LIN {X 0,Y 256.268,Z 255.065,A -85,B 0,C 180,E1 -18646.324,E2 -18646.324} C_VEL
LIN {X 0,Y 256.169,Z 255.063,A -85,B 0,C 180,E1 -18651.153,E2 -18651.153} C_VEL
LIN {X 0,Y 256.159,Z 255.045,A -85,B 0,C 180,E1 -18655.146,E2 -18655.146} C_VEL
LIN {X 0,Y 256.122,Z 255.064,A -85,B 0,C 180,E1 -18659.598,E2 -18659.598} C_VEL
LIN {X 0,Y 256.095,Z 255.082,A -85,B 0,C 180,E1 -18663.288,E2 -18663.288} C_VEL
LIN {X 0,Y 256.131,Z 255.076,A -85,B 0,C 180,E1 -18667.291,E2 -18667.291} C_VEL
LIN {X 0,Y 256.137,Z 255.062,A -85,B 0,C 180,E1 -18671.186,E2 -18671.186} C_VEL
LIN {X 0,Y 256.089,Z 255.082,A -85,B 0,C 180,E1 -18675.522,E2 -18675.522} C_VEL
LIN {X 0,Y 256.106,Z 255.073,A -85,B 0,C 180,E1 -18678.818,E2 -18678.818} C_VEL
LIN {X 0,Y 256.13,Z 255.056,A -85,B 0,C 180,E1 -18682.878,E2 -18682.878} C_VEL
LIN {X 0,Y 256.062,Z 255.088,A -85,B 0,C 180,E1 -18686.717,E2 -18686.717} C_VEL
LIN {X 0,Y 256.118,Z 255.044,A -85,B 0,C 180,E1 -18691.412,E2 -18691.412} C_VEL
LIN {X 0,Y 256.151,Z 255.067,A -85,B 0,C 180,E1 -18695.706,E2 -18695.706} C_VEL
LIN {X 0,Y 256.218,Z 255.067,A -85,B 0,C 180,E1 -18699.118,E2 -18699.118} C_VEL
LIN {X 0,Y 256.282,Z 255.016,A -85,B 0,C 180,E1 -18704.092,E2 -18704.092} C_VEL
LIN {X 0,Y 256.301,Z 255.048,A -85,B 0,C 180,E1 -18708.941,E2 -18708.941} C_VEL
LIN {X 0,Y 256.533,Z 255.027,A -85,B 0,C 180,E1 -18712.134,E2 -18712.134} C_VEL
LIN {X 0,Y 256.71,Z 254.962,A -85,B 0,C 180,E1 -18718.438,E2 -18718.438} C_VEL
LIN {X 0,Y 256.736,Z 254.971,A -85,B 0,C 180,E1 -18719.772,E2 -18719.772} C_VEL
LIN {X 0,Y 256.465,Z 255.019,A -85,B 0,C 180,E1 -18720.645,E2 -18720.645} C_VEL
LIN {X 0,Y 255.123,Z 255.201,A -85,B 0,C 180,E1 -18721.933,E2 -18721.933} C_VEL
LIN {X 0,Y 250.65,Z 255.767,A -85,B 0,C 180,E1 -18724.929,E2 -18724.929} C_VEL
LIN {X 0,Y 249.524,Z 255.896,A -85,B 0,C 180,E1 -18726.273,E2 -18726.273} C_VEL
LIN {X 0,Y 249.417,Z 255.903,A -85,B 0,C 180,E1 -18726.73,E2 -18726.73} C_VEL
LIN {X 0,Y 249.345,Z 255.885,A -85,B 0,C 180,E1 -18729.743,E2 -18729.743} C_VEL
LIN {X 0,Y 249.21,Z 255.942,A -85,B 0,C 180,E1 -18734.71,E2 -18734.71} C_VEL
LIN {X 0,Y 249.144,Z 255.941,A -85,B 0,C 180,E1 -18738.084,E2 -18738.084} C_VEL
LIN {X 0,Y 249.091,Z 255.926,A -85,B 0,C 180,E1 -18741.524,E2 -18741.524} C_VEL
LIN {X 0,Y 249.125,Z 255.954,A -85,B 0,C 180,E1 -18745.481,E2 -18745.481} C_VEL
LIN {X 0,Y 249.065,Z 255.939,A -85,B 0,C 180,E1 -18748.987,E2 -18748.987} C_VEL
LIN {X 0,Y 249.038,Z 255.962,A -85,B 0,C 180,E1 -18752.432,E2 -18752.432} C_VEL
LIN {X 0,Y 249.038,Z 255.952,A -85,B 0,C 180,E1 -18756.351,E2 -18756.351} C_VEL
LIN {X 0,Y 249.019,Z 255.966,A -85,B 0,C 180,E1 -18760.483,E2 -18760.483} C_VEL
LIN {X 0,Y 249.014,Z 255.942,A -85,B 0,C 180,E1 -18762.795,E2 -18762.795} C_VEL
LIN {X 0,Y 248.992,Z 255.944,A -85,B 0,C 180,E1 -18767.359,E2 -18767.359} C_VEL
LIN {X 0,Y 249.017,Z 255.952,A -85,B 0,C 180,E1 -18771.619,E2 -18771.619} C_VEL
LIN {X 0,Y 249.109,Z 256,A -85,B 0,C 180,E1 -18776.504,E2 -18776.504} C_VEL
LIN {X 0,Y 251.031,Z 265.205,A -85,B 0,C 180,E1 -18780.224,E2 -18780.224} C_VEL
LIN {X 0,Y 251.514,Z 267.303,A -85,B 0,C 180,E1 -18780.91,E2 -18780.91} C_VEL
LIN {X 0,Y 257.248,Z 283.893,A -85,B 0,C 180,E1 -18782.001,E2 -18782.001} C_VEL
LIN {X 0,Y 261.027,Z 311.595,A -85,B 0,C 180,E1 -18783.167,E2 -18783.167} C_VEL
LIN {X 0,Y 259.211,Z 375.113,A -85,B 0,C 180,E1 -18784.936,E2 -18784.936} C_VEL
LIN {X 0,Y 258.333,Z 387.52,A -85,B 0,C 180,E1 -18785.543,E2 -18785.543} C_VEL
LIN {X 0,Y 257.11,Z 401.037,A -85,B 0,C 180,E1 -18786.544,E2 -18786.544} C_VEL
LIN {X 0,Y 255.546,Z 413.128,A -85,B 0,C 180,E1 -18787.781,E2 -18787.781} C_VEL
LIN {X 0,Y 253.899,Z 424.693,A -85,B 0,C 180,E1 -18789.334,E2 -18789.334} C_VEL
LIN {X 0,Y 252.383,Z 435.261,A -85,B 0,C 180,E1 -18791.141,E2 -18791.141} C_VEL
LIN {X 0,Y 250.81,Z 445.277,A -85,B 0,C 180,E1 -18793.309,E2 -18793.309} C_VEL
LIN {X 0,Y 249.345,Z 454.181,A -85,B 0,C 180,E1 -18795.723,E2 -18795.723} C_VEL
LIN {X 0,Y 248.261,Z 461.278,A -85,B 0,C 180,E1 -18798.157,E2 -18798.157} C_VEL
LIN {X 0,Y 247.426,Z 467.749,A -85,B 0,C 180,E1 -18801.013,E2 -18801.013} C_VEL
LIN {X 0,Y 247.028,Z 471.99,A -85,B 0,C 180,E1 -18803.466,E2 -18803.466} C_VEL
LIN {X 0,Y 246.86,Z 474.371,A -85,B 0,C 180,E1 -18805.217,E2 -18805.217} C_VEL
LIN {X 0,Y 246.839,Z 475.983,A -85,B 0,C 180,E1 -18806.736,E2 -18806.736} C_VEL
LIN {X 0,Y 246.87,Z 477.31,A -85,B 0,C 180,E1 -18808.369,E2 -18808.369} C_VEL
LIN {X 0,Y 246.903,Z 478.239,A -85,B 0,C 180,E1 -18810.001,E2 -18810.001} C_VEL
LIN {X 0,Y 246.87,Z 478.771,A -85,B 0,C 180,E1 -18811.632,E2 -18811.632} C_VEL
LIN {X 0,Y 246.942,Z 478.586,A -85,B 0,C 180,E1 -18814.898,E2 -18814.898} C_VEL
LIN {X 0,Y 247.422,Z 476.873,A -85,B 0,C 180,E1 -18818.166,E2 -18818.166} C_VEL
LIN {X 0,Y 247.888,Z 475.394,A -85,B 0,C 180,E1 -18819.795,E2 -18819.795} C_VEL
LIN {X 0,Y 248.918,Z 472.402,A -85,B 0,C 180,E1 -18822.226,E2 -18822.226} C_VEL
LIN {X 0,Y 250.251,Z 468.389,A -85,B 0,C 180,E1 -18824.641,E2 -18824.641} C_VEL
LIN {X 0,Y 252.491,Z 462.242,A -85,B 0,C 180,E1 -18827.411,E2 -18827.411} C_VEL
LIN {X 0,Y 254.814,Z 455.623,A -85,B 0,C 180,E1 -18829.73,E2 -18829.73} C_VEL
LIN {X 0,Y 257.32,Z 447.491,A -85,B 0,C 180,E1 -18832.016,E2 -18832.016} C_VEL
LIN {X 0,Y 259.942,Z 438.896,A -85,B 0,C 180,E1 -18833.926,E2 -18833.926} C_VEL
LIN {X 0,Y 262.902,Z 428.491,A -85,B 0,C 180,E1 -18835.748,E2 -18835.748} C_VEL
LIN {X 0,Y 265.736,Z 416.819,A -85,B 0,C 180,E1 -18837.357,E2 -18837.357} C_VEL
LIN {X 0,Y 268.156,Z 405.109,A -85,B 0,C 180,E1 -18838.575,E2 -18838.575} C_VEL
LIN {X 0,Y 270.132,Z 393.004,A -85,B 0,C 180,E1 -18839.518,E2 -18839.518} C_VEL
LIN {X 0,Y 271.689,Z 379.85,A -85,B 0,C 180,E1 -18840.239,E2 -18840.239} C_VEL
LIN {X 0,Y 272.619,Z 364.907,A -85,B 0,C 180,E1 -18840.726,E2 -18840.726} C_VEL
LIN {X 0,Y 274.682,Z 317.162,A -85,B 0,C 180,E1 -18841.977,E2 -18841.977} C_VEL
LIN {X 0,Y 272.652,Z 306.034,A -85,B 0,C 180,E1 -18842.686,E2 -18842.686} C_VEL
LIN {X 0,Y 266.598,Z 292.603,A -85,B 0,C 180,E1 -18844.214,E2 -18844.214} C_VEL
LIN {X 0,Y 257.687,Z 275.866,A -85,B 0,C 180,E1 -18846.542,E2 -18846.542} C_VEL
LIN {X 0,Y 254.296,Z 270.358,A -85,B 0,C 180,E1 -18847.462,E2 -18847.462} C_VEL
LIN {X 0,Y 251.99,Z 266.272,A -85,B 0,C 180,E1 -18848.205,E2 -18848.205} C_VEL
LIN {X 0,Y 249.946,Z 259.327,A -85,B 0,C 180,E1 -18851.822,E2 -18851.822} C_VEL
LIN {X 0,Y 249.003,Z 255.983,A -85,B 0,C 180,E1 -18853.876,E2 -18853.876} C_VEL
LIN {X 0,Y 249.022,Z 255.94,A -85,B 0,C 180,E1 -18857.357,E2 -18857.357} C_VEL
LIN {X 0,Y 249.056,Z 255.957,A -85,B 0,C 180,E1 -18862.197,E2 -18862.197} C_VEL
LIN {X 0,Y 249.058,Z 255.959,A -85,B 0,C 180,E1 -18865.635,E2 -18865.635} C_VEL
LIN {X 0,Y 249.015,Z 255.966,A -85,B 0,C 180,E1 -18869.461,E2 -18869.461} C_VEL
LIN {X 0,Y 249.028,Z 255.962,A -85,B 0,C 180,E1 -18873.15,E2 -18873.15} C_VEL
LIN {X 0,Y 249.017,Z 255.959,A -85,B 0,C 180,E1 -18876.72,E2 -18876.72} C_VEL
LIN {X 0,Y 249.068,Z 255.947,A -85,B 0,C 180,E1 -18880.201,E2 -18880.201} C_VEL
LIN {X 0,Y 249.186,Z 255.935,A -85,B 0,C 180,E1 -18883.611,E2 -18883.611} C_VEL
LIN {X 0,Y 249.245,Z 255.926,A -85,B 0,C 180,E1 -18888.609,E2 -18888.609} C_VEL
LIN {X 0,Y 249.445,Z 255.913,A -85,B 0,C 180,E1 -18891.895,E2 -18891.895} C_VEL
LIN {X 0,Y 249.277,Z 255.928,A -85,B 0,C 180,E1 -18895.141,E2 -18895.141} C_VEL
LIN {X 0,Y 249.666,Z 255.872,A -85,B 0,C 180,E1 -18898.38,E2 -18898.38} C_VEL
LIN {X 0,Y 249.671,Z 255.881,A -85,B 0,C 180,E1 -18901.606,E2 -18901.606} C_VEL
LIN {X 0,Y 249.425,Z 255.906,A -85,B 0,C 180,E1 -18906.532,E2 -18906.532} C_VEL
LIN {X 0,Y 249.34,Z 255.927,A -85,B 0,C 180,E1 -18909.729,E2 -18909.729} C_VEL
LIN {X 0,Y 249.176,Z 255.939,A -85,B 0,C 180,E1 -18914.697,E2 -18914.697} C_VEL
LIN {X 0,Y 249.111,Z 255.949,A -85,B 0,C 180,E1 -18918.071,E2 -18918.071} C_VEL
LIN {X 0,Y 249.076,Z 255.953,A -85,B 0,C 180,E1 -18921.51,E2 -18921.51} C_VEL
LIN {X 0,Y 249.116,Z 255.93,A -85,B 0,C 180,E1 -18925.474,E2 -18925.474} C_VEL
LIN {X 0,Y 249.033,Z 255.949,A -85,B 0,C 180,E1 -18930.095,E2 -18930.095} C_VEL
LIN {X 0,Y 249.056,Z 256.275,A -85,B 0,C 180,E1 -18930.751,E2 -18930.751} C_VEL
LIN {X 0,Y 250.702,Z 261.422,A -85,B 0,C 180,E1 -18933.56,E2 -18933.56} C_VEL
LIN {X 0,Y 253.421,Z 265.892,A -85,B 0,C 180,E1 -18934.408,E2 -18934.408} C_VEL
LIN {X 0,Y 259.859,Z 276.539,A -85,B 0,C 180,E1 -18936.154,E2 -18936.154} C_VEL
LIN {X 0,Y 266.04,Z 287.62,A -85,B 0,C 180,E1 -18937.741,E2 -18937.741} C_VEL
LIN {X 0,Y 273.058,Z 302.502,A -85,B 0,C 180,E1 -18939.498,E2 -18939.498} C_VEL
LIN {X 0,Y 275.043,Z 307.322,A -85,B 0,C 180,E1 -18939.99,E2 -18939.99} C_VEL
LIN {X 0,Y 272.309,Z 368.99,A -85,B 0,C 180,E1 -18941.647,E2 -18941.647} C_VEL
LIN {X 0,Y 271.045,Z 381.678,A -85,B 0,C 180,E1 -18942.233,E2 -18942.233} C_VEL
LIN {X 0,Y 269.395,Z 393.837,A -85,B 0,C 180,E1 -18943.074,E2 -18943.074} C_VEL
LIN {X 0,Y 267.158,Z 405.932,A -85,B 0,C 180,E1 -18944.204,E2 -18944.204} C_VEL
LIN {X 0,Y 264.797,Z 416.671,A -85,B 0,C 180,E1 -18945.531,E2 -18945.531} C_VEL
LIN {X 0,Y 261.869,Z 428.103,A -85,B 0,C 180,E1 -18947.339,E2 -18947.339} C_VEL
LIN {X 0,Y 258.942,Z 438.019,A -85,B 0,C 180,E1 -18949.353,E2 -18949.353} C_VEL
LIN {X 0,Y 256.367,Z 446.072,A -85,B 0,C 180,E1 -18951.415,E2 -18951.415} C_VEL
LIN {X 0,Y 253.816,Z 453.448,A -85,B 0,C 180,E1 -18953.782,E2 -18953.782} C_VEL
LIN {X 0,Y 251.804,Z 459.061,A -85,B 0,C 180,E1 -18956.067,E2 -18956.067} C_VEL
LIN {X 0,Y 249.967,Z 464.011,A -85,B 0,C 180,E1 -18958.658,E2 -18958.658} C_VEL
LIN {X 0,Y 248.598,Z 467.684,A -85,B 0,C 180,E1 -18961.275,E2 -18961.275} C_VEL
LIN {X 0,Y 247.898,Z 469.469,A -85,B 0,C 180,E1 -18963.024,E2 -18963.024} C_VEL
LIN {X 0,Y 247.242,Z 471.174,A -85,B 0,C 180,E1 -18965.429,E2 -18965.429} C_VEL
LIN {X 0,Y 246.716,Z 472.063,A -85,B 0,C 180,E1 -18968.264,E2 -18968.264} C_VEL
LIN {X 0,Y 246.593,Z 472.02,A -85,B 0,C 180,E1 -18970.109,E2 -18970.109} C_VEL
LIN {X 0,Y 246.5,Z 471.576,A -85,B 0,C 180,E1 -18971.722,E2 -18971.722} C_VEL
LIN {X 0,Y 246.481,Z 470.644,A -85,B 0,C 180,E1 -18973.433,E2 -18973.433} C_VEL
LIN {X 0,Y 246.665,Z 468.876,A -85,B 0,C 180,E1 -18975.594,E2 -18975.594} C_VEL
LIN {X 0,Y 247.089,Z 465.228,A -85,B 0,C 180,E1 -18978.515,E2 -18978.515} C_VEL
LIN {X 0,Y 247.589,Z 460.912,A -85,B 0,C 180,E1 -18981.018,E2 -18981.018} C_VEL
LIN {X 0,Y 248.411,Z 455.369,A -85,B 0,C 180,E1 -18983.502,E2 -18983.502} C_VEL
LIN {X 0,Y 249.424,Z 448.448,A -85,B 0,C 180,E1 -18985.96,E2 -18985.96} C_VEL
LIN {X 0,Y 250.55,Z 441.374,A -85,B 0,C 180,E1 -18987.99,E2 -18987.99} C_VEL
LIN {X 0,Y 251.912,Z 432.846,A -85,B 0,C 180,E1 -18989.999,E2 -18989.999} C_VEL
LIN {X 0,Y 253.636,Z 422.254,A -85,B 0,C 180,E1 -18991.984,E2 -18991.984} C_VEL
LIN {X 0,Y 255.344,Z 410.323,A -85,B 0,C 180,E1 -18993.747,E2 -18993.747} C_VEL
LIN {X 0,Y 256.801,Z 398.302,A -85,B 0,C 180,E1 -18995.102,E2 -18995.102} C_VEL
LIN {X 0,Y 257.943,Z 385.834,A -85,B 0,C 180,E1 -18996.158,E2 -18996.158} C_VEL
LIN {X 0,Y 258.952,Z 372.79,A -85,B 0,C 180,E1 -18996.917,E2 -18996.917} C_VEL
LIN {X 0,Y 259.526,Z 357.393,A -85,B 0,C 180,E1 -18997.439,E2 -18997.439} C_VEL
LIN {X 0,Y 261.24,Z 299.46,A -85,B 0,C 180,E1 -18999.006,E2 -18999.006} C_VEL
LIN {X 0,Y 259.014,Z 285.584,A -85,B 0,C 180,E1 -18999.617,E2 -18999.617} C_VEL
LIN {X 0,Y 253.614,Z 269.571,A -85,B 0,C 180,E1 -19000.609,E2 -19000.609} C_VEL
LIN {X 0,Y 250.347,Z 261.084,A -85,B 0,C 180,E1 -19001.239,E2 -19001.239} C_VEL
LIN {X 0,Y 249.257,Z 256.073,A -85,B 0,C 180,E1 -19003.191,E2 -19003.191} C_VEL
LIN {X 0,Y 249.21,Z 255.943,A -85,B 0,C 180,E1 -19006.531,E2 -19006.531} C_VEL
LIN {X 0,Y 249.103,Z 255.948,A -85,B 0,C 180,E1 -19011.516,E2 -19011.516} C_VEL
LIN {X 0,Y 249.1,Z 255.918,A -85,B 0,C 180,E1 -19015.489,E2 -19015.489} C_VEL
LIN {X 0,Y 249.099,Z 255.929,A -85,B 0,C 180,E1 -19019.019,E2 -19019.019} C_VEL
LIN {X 0,Y 249.039,Z 255.966,A -85,B 0,C 180,E1 -19022.424,E2 -19022.424} C_VEL
LIN {X 0,Y 249.061,Z 255.95,A -85,B 0,C 180,E1 -19026.339,E2 -19026.339} C_VEL
LIN {X 0,Y 249.104,Z 255.947,A -85,B 0,C 180,E1 -19030.458,E2 -19030.458} C_VEL
LIN {X 0,Y 249.035,Z 255.959,A -85,B 0,C 180,E1 -19034.871,E2 -19034.871} C_VEL
LIN {X 0,Y 249.071,Z 255.959,A -85,B 0,C 180,E1 -19037.387,E2 -19037.387} C_VEL
LIN {X 0,Y 249.027,Z 255.931,A -85,B 0,C 180,E1 -19041.631,E2 -19041.631} C_VEL
LIN {X 0,Y 249.038,Z 255.961,A -85,B 0,C 180,E1 -19045.649,E2 -19045.649} C_VEL
LIN {X 0,Y 249.031,Z 255.95,A -85,B 0,C 180,E1 -19049.48,E2 -19049.48} C_VEL
LIN {X 0,Y 249.055,Z 255.922,A -85,B 0,C 180,E1 -19053.17,E2 -19053.17} C_VEL
LIN {X 0,Y 249.071,Z 255.954,A -85,B 0,C 180,E1 -19056.741,E2 -19056.741} C_VEL
LIN {X 0,Y 249.132,Z 255.948,A -85,B 0,C 180,E1 -19060.222,E2 -19060.222} C_VEL
LIN {X 0,Y 249.23,Z 255.897,A -85,B 0,C 180,E1 -19063.629,E2 -19063.629} C_VEL
LIN {X 0,Y 249.244,Z 255.925,A -85,B 0,C 180,E1 -19068.624,E2 -19068.624} C_VEL
LIN {X 0,Y 249.477,Z 255.906,A -85,B 0,C 180,E1 -19071.91,E2 -19071.91} C_VEL
LIN {X 0,Y 249.43,Z 255.871,A -85,B 0,C 180,E1 -19076.777,E2 -19076.777} C_VEL
LIN {X 0,Y 249.718,Z 255.848,A -85,B 0,C 180,E1 -19080.007,E2 -19080.007} C_VEL
LIN {X 0,Y 249.43,Z 255.912,A -85,B 0,C 180,E1 -19083.238,E2 -19083.238} C_VEL
LIN {X 0,Y 249.417,Z 255.903,A -85,B 0,C 180,E1 -19086.73,E2 -19086.73} C_VEL
LIN {X 0,Y 248.696,Z 255.981,A -85,B 0,C 180,E1 -19088.076,E2 -19088.076} C_VEL
LIN {X 0,Y 245.771,Z 256.344,A -85,B 0,C 180,E1 -19090.268,E2 -19090.268} C_VEL
LIN {X 0,Y 243.304,Z 256.66,A -85,B 0,C 180,E1 -19092.054,E2 -19092.054} C_VEL
LIN {X 0,Y 242.237,Z 256.8,A -85,B 0,C 180,E1 -19093.441,E2 -19093.441} C_VEL
LIN {X 0,Y 242.145,Z 256.811,A -85,B 0,C 180,E1 -19093.911,E2 -19093.911} C_VEL
LIN {X 0,Y 242.156,Z 256.818,A -85,B 0,C 180,E1 -19096.878,E2 -19096.878} C_VEL
LIN {X 0,Y 242.033,Z 256.806,A -85,B 0,C 180,E1 -19101.693,E2 -19101.693} C_VEL
LIN {X 0,Y 242.076,Z 256.832,A -85,B 0,C 180,E1 -19105.844,E2 -19105.844} C_VEL
LIN {X 0,Y 241.986,Z 256.818,A -85,B 0,C 180,E1 -19109.593,E2 -19109.593} C_VEL
LIN {X 0,Y 241.99,Z 256.846,A -85,B 0,C 180,E1 -19113.498,E2 -19113.498} C_VEL
LIN {X 0,Y 241.995,Z 256.826,A -85,B 0,C 180,E1 -19117.588,E2 -19117.588} C_VEL
LIN {X 0,Y 241.947,Z 256.838,A -85,B 0,C 180,E1 -19121.928,E2 -19121.928} C_VEL
LIN {X 0,Y 241.916,Z 256.811,A -85,B 0,C 180,E1 -19126.584,E2 -19126.584} C_VEL
LIN {X 0,Y 241.944,Z 256.844,A -85,B 0,C 180,E1 -19130.28,E2 -19130.28} C_VEL
LIN {X 0,Y 241.989,Z 256.841,A -85,B 0,C 180,E1 -19134.49,E2 -19134.49} C_VEL
LIN {X 0,Y 242.088,Z 257.038,A -85,B 0,C 180,E1 -19136.15,E2 -19136.15} C_VEL
LIN {X 0,Y 244.179,Z 266.965,A -85,B 0,C 180,E1 -19140.133,E2 -19140.133} C_VEL
LIN {X 0,Y 246.952,Z 274.593,A -85,B 0,C 180,E1 -19140.729,E2 -19140.729} C_VEL
LIN {X 0,Y 250.974,Z 286.669,A -85,B 0,C 180,E1 -19141.497,E2 -19141.497} C_VEL
LIN {X 0,Y 254.446,Z 312.616,A -85,B 0,C 180,E1 -19142.618,E2 -19142.618} C_VEL
LIN {X 0,Y 252.549,Z 374.939,A -85,B 0,C 180,E1 -19144.393,E2 -19144.393} C_VEL
LIN {X 0,Y 251.653,Z 387.375,A -85,B 0,C 180,E1 -19145.014,E2 -19145.014} C_VEL
LIN {X 0,Y 250.447,Z 400.339,A -85,B 0,C 180,E1 -19145.991,E2 -19145.991} C_VEL
LIN {X 0,Y 248.968,Z 411.809,A -85,B 0,C 180,E1 -19147.162,E2 -19147.162} C_VEL
LIN {X 0,Y 247.192,Z 423.597,A -85,B 0,C 180,E1 -19148.747,E2 -19148.747} C_VEL
LIN {X 0,Y 245.658,Z 434.253,A -85,B 0,C 180,E1 -19150.584,E2 -19150.584} C_VEL
LIN {X 0,Y 244.328,Z 442.864,A -85,B 0,C 180,E1 -19152.421,E2 -19152.421} C_VEL
LIN {X 0,Y 242.933,Z 450.808,A -85,B 0,C 180,E1 -19154.479,E2 -19154.479} C_VEL
LIN {X 0,Y 241.563,Z 458.535,A -85,B 0,C 180,E1 -19156.97,E2 -19156.97} C_VEL
LIN {X 0,Y 240.842,Z 463.824,A -85,B 0,C 180,E1 -19159.067,E2 -19159.067} C_VEL
LIN {X 0,Y 240.224,Z 468.923,A -85,B 0,C 180,E1 -19161.589,E2 -19161.589} C_VEL
LIN {X 0,Y 239.847,Z 472.858,A -85,B 0,C 180,E1 -19164.114,E2 -19164.114} C_VEL
LIN {X 0,Y 239.746,Z 475.746,A -85,B 0,C 180,E1 -19166.639,E2 -19166.639} C_VEL
LIN {X 0,Y 239.784,Z 477.105,A -85,B 0,C 180,E1 -19168.321,E2 -19168.321} C_VEL
LIN {X 0,Y 239.816,Z 478.064,A -85,B 0,C 180,E1 -19170.001,E2 -19170.001} C_VEL
LIN {X 0,Y 239.784,Z 478.631,A -85,B 0,C 180,E1 -19171.68,E2 -19171.68} C_VEL
LIN {X 0,Y 239.855,Z 478.57,A -85,B 0,C 180,E1 -19174.916,E2 -19174.916} C_VEL
LIN {X 0,Y 240.055,Z 477.898,A -85,B 0,C 180,E1 -19176.726,E2 -19176.726} C_VEL
LIN {X 0,Y 240.894,Z 475.469,A -85,B 0,C 180,E1 -19180.082,E2 -19180.082} C_VEL
LIN {X 0,Y 241.975,Z 472.536,A -85,B 0,C 180,E1 -19182.582,E2 -19182.582} C_VEL
LIN {X 0,Y 243.372,Z 468.589,A -85,B 0,C 180,E1 -19185.065,E2 -19185.065} C_VEL
LIN {X 0,Y 245.398,Z 463.528,A -85,B 0,C 180,E1 -19187.501,E2 -19187.501} C_VEL
LIN {X 0,Y 247.768,Z 457.187,A -85,B 0,C 180,E1 -19189.901,E2 -19189.901} C_VEL
LIN {X 0,Y 250.209,Z 449.606,A -85,B 0,C 180,E1 -19192.197,E2 -19192.197} C_VEL
LIN {X 0,Y 252.952,Z 441.298,A -85,B 0,C 180,E1 -19194.193,E2 -19194.193} C_VEL
LIN {X 0,Y 255.966,Z 431.541,A -85,B 0,C 180,E1 -19196.06,E2 -19196.06} C_VEL
LIN {X 0,Y 258.874,Z 420.66,A -85,B 0,C 180,E1 -19197.705,E2 -19197.705} C_VEL
LIN {X 0,Y 261.315,Z 410.047,A -85,B 0,C 180,E1 -19198.954,E2 -19198.954} C_VEL
LIN {X 0,Y 263.489,Z 398.442,A -85,B 0,C 180,E1 -19200.008,E2 -19200.008} C_VEL
LIN {X 0,Y 265.39,Z 385.352,A -85,B 0,C 180,E1 -19200.867,E2 -19200.867} C_VEL
LIN {X 0,Y 266.579,Z 372.119,A -85,B 0,C 180,E1 -19201.427,E2 -19201.427} C_VEL
LIN {X 0,Y 269.08,Z 318.313,A -85,B 0,C 180,E1 -19202.874,E2 -19202.874} C_VEL
LIN {X 0,Y 267.46,Z 309.167,A -85,B 0,C 180,E1 -19203.475,E2 -19203.475} C_VEL
LIN {X 0,Y 261.518,Z 296.019,A -85,B 0,C 180,E1 -19205.04,E2 -19205.04} C_VEL
LIN {X 0,Y 253.419,Z 280.618,A -85,B 0,C 180,E1 -19207.254,E2 -19207.254} C_VEL
LIN {X 0,Y 249.605,Z 274.39,A -85,B 0,C 180,E1 -19208.34,E2 -19208.34} C_VEL
LIN {X 0,Y 247.069,Z 270.251,A -85,B 0,C 180,E1 -19209.102,E2 -19209.102} C_VEL
LIN {X 0,Y 244.678,Z 266.104,A -85,B 0,C 180,E1 -19209.931,E2 -19209.931} C_VEL
LIN {X 0,Y 242.716,Z 259.494,A -85,B 0,C 180,E1 -19213.615,E2 -19213.615} C_VEL
LIN {X 0,Y 241.944,Z 256.873,A -85,B 0,C 180,E1 -19215.396,E2 -19215.396} C_VEL
LIN {X 0,Y 241.935,Z 256.835,A -85,B 0,C 180,E1 -19219.05,E2 -19219.05} C_VEL
LIN {X 0,Y 241.999,Z 256.838,A -85,B 0,C 180,E1 -19222.413,E2 -19222.413} C_VEL
LIN {X 0,Y 241.994,Z 256.843,A -85,B 0,C 180,E1 -19226.502,E2 -19226.502} C_VEL
LIN {X 0,Y 241.989,Z 256.837,A -85,B 0,C 180,E1 -19230.608,E2 -19230.608} C_VEL
LIN {X 0,Y 242.008,Z 256.839,A -85,B 0,C 180,E1 -19234.192,E2 -19234.192} C_VEL
LIN {X 0,Y 241.997,Z 256.841,A -85,B 0,C 180,E1 -19238.332,E2 -19238.332} C_VEL
LIN {X 0,Y 242.125,Z 256.817,A -85,B 0,C 180,E1 -19243.31,E2 -19243.31} C_VEL
LIN {X 0,Y 242.18,Z 256.808,A -85,B 0,C 180,E1 -19248.272,E2 -19248.272} C_VEL
LIN {X 0,Y 242.394,Z 256.793,A -85,B 0,C 180,E1 -19251.657,E2 -19251.657} C_VEL
LIN {X 0,Y 242.238,Z 256.803,A -85,B 0,C 180,E1 -19254.999,E2 -19254.999} C_VEL
LIN {X 0,Y 242.625,Z 256.749,A -85,B 0,C 180,E1 -19258.333,E2 -19258.333} C_VEL
LIN {X 0,Y 242.632,Z 256.757,A -85,B 0,C 180,E1 -19261.652,E2 -19261.652} C_VEL
LIN {X 0,Y 242.399,Z 256.78,A -85,B 0,C 180,E1 -19266.652,E2 -19266.652} C_VEL
LIN {X 0,Y 242.264,Z 256.805,A -85,B 0,C 180,E1 -19270.016,E2 -19270.016} C_VEL
LIN {X 0,Y 242.132,Z 256.814,A -85,B 0,C 180,E1 -19275.135,E2 -19275.135} C_VEL
LIN {X 0,Y 242.05,Z 256.826,A -85,B 0,C 180,E1 -19278.617,E2 -19278.617} C_VEL
LIN {X 0,Y 242.001,Z 256.833,A -85,B 0,C 180,E1 -19282.172,E2 -19282.172} C_VEL
LIN {X 0,Y 242.053,Z 256.807,A -85,B 0,C 180,E1 -19285.83,E2 -19285.83} C_VEL
LIN {X 0,Y 242.05,Z 256.877,A -85,B 0,C 180,E1 -19289.008,E2 -19289.008} C_VEL
LIN {X 0,Y 243.33,Z 261.381,A -85,B 0,C 180,E1 -19291.739,E2 -19291.739} C_VEL
LIN {X 0,Y 245.842,Z 265.498,A -85,B 0,C 180,E1 -19292.639,E2 -19292.639} C_VEL
LIN {X 0,Y 252.53,Z 275.938,A -85,B 0,C 180,E1 -19294.607,E2 -19294.607} C_VEL
LIN {X 0,Y 260.166,Z 289.495,A -85,B 0,C 180,E1 -19296.693,E2 -19296.693} C_VEL
LIN {X 0,Y 266.617,Z 302.832,A -85,B 0,C 180,E1 -19298.386,E2 -19298.386} C_VEL
LIN {X 0,Y 269.412,Z 309.425,A -85,B 0,C 180,E1 -19299.111,E2 -19299.111} C_VEL
LIN {X 0,Y 266.606,Z 369.315,A -85,B 0,C 180,E1 -19300.752,E2 -19300.752} C_VEL
LIN {X 0,Y 265.275,Z 382.204,A -85,B 0,C 180,E1 -19301.365,E2 -19301.365} C_VEL
LIN {X 0,Y 263.469,Z 394.658,A -85,B 0,C 180,E1 -19302.249,E2 -19302.249} C_VEL
LIN {X 0,Y 261.148,Z 406.518,A -85,B 0,C 180,E1 -19303.396,E2 -19303.396} C_VEL
LIN {X 0,Y 258.299,Z 418.736,A -85,B 0,C 180,E1 -19304.974,E2 -19304.974} C_VEL
LIN {X 0,Y 255.324,Z 429.583,A -85,B 0,C 180,E1 -19306.787,E2 -19306.787} C_VEL
LIN {X 0,Y 252.236,Z 439.422,A -85,B 0,C 180,E1 -19308.893,E2 -19308.893} C_VEL
LIN {X 0,Y 249.411,Z 447.817,A -85,B 0,C 180,E1 -19311.173,E2 -19311.173} C_VEL
LIN {X 0,Y 246.647,Z 455.225,A -85,B 0,C 180,E1 -19313.754,E2 -19313.754} C_VEL
LIN {X 0,Y 244.277,Z 461.337,A -85,B 0,C 180,E1 -19316.531,E2 -19316.531} C_VEL
LIN {X 0,Y 242.37,Z 466.176,A -85,B 0,C 180,E1 -19319.506,E2 -19319.506} C_VEL
LIN {X 0,Y 241.095,Z 469.234,A -85,B 0,C 180,E1 -19322.198,E2 -19322.198} C_VEL
LIN {X 0,Y 240.228,Z 471.271,A -85,B 0,C 180,E1 -19325.06,E2 -19325.06} C_VEL
LIN {X 0,Y 239.716,Z 472.129,A -85,B 0,C 180,E1 -19327.596,E2 -19327.596} C_VEL
LIN {X 0,Y 239.498,Z 472.124,A -85,B 0,C 180,E1 -19329.86,E2 -19329.86} C_VEL
LIN {X 0,Y 239.375,Z 471.003,A -85,B 0,C 180,E1 -19332.926,E2 -19332.926} C_VEL
LIN {X 0,Y 239.565,Z 469.06,A -85,B 0,C 180,E1 -19335.449,E2 -19335.449} C_VEL
LIN {X 0,Y 239.935,Z 465.888,A -85,B 0,C 180,E1 -19338.168,E2 -19338.168} C_VEL
LIN {X 0,Y 240.405,Z 461.74,A -85,B 0,C 180,E1 -19340.747,E2 -19340.747} C_VEL
LIN {X 0,Y 241.391,Z 455.34,A -85,B 0,C 180,E1 -19343.731,E2 -19343.731} C_VEL
LIN {X 0,Y 242.436,Z 448.393,A -85,B 0,C 180,E1 -19346.26,E2 -19346.26} C_VEL
LIN {X 0,Y 243.619,Z 441.287,A -85,B 0,C 180,E1 -19348.346,E2 -19348.346} C_VEL
LIN {X 0,Y 245.071,Z 432.517,A -85,B 0,C 180,E1 -19350.451,E2 -19350.451} C_VEL
LIN {X 0,Y 246.862,Z 421.841,A -85,B 0,C 180,E1 -19352.483,E2 -19352.483} C_VEL
LIN {X 0,Y 248.606,Z 410.037,A -85,B 0,C 180,E1 -19354.255,E2 -19354.255} C_VEL
LIN {X 0,Y 250.112,Z 397.885,A -85,B 0,C 180,E1 -19355.643,E2 -19355.643} C_VEL
LIN {X 0,Y 251.29,Z 385.26,A -85,B 0,C 180,E1 -19356.725,E2 -19356.725} C_VEL
LIN {X 0,Y 252.281,Z 372.846,A -85,B 0,C 180,E1 -19357.452,E2 -19357.452} C_VEL
LIN {X 0,Y 252.876,Z 357.439,A -85,B 0,C 180,E1 -19357.987,E2 -19357.987} C_VEL
LIN {X 0,Y 254.641,Z 299.96,A -85,B 0,C 180,E1 -19359.581,E2 -19359.581} C_VEL
LIN {X 0,Y 252.6,Z 287.557,A -85,B 0,C 180,E1 -19360.152,E2 -19360.152} C_VEL
LIN {X 0,Y 247.577,Z 272.582,A -85,B 0,C 180,E1 -19361.115,E2 -19361.115} C_VEL
LIN {X 0,Y 243.17,Z 261.277,A -85,B 0,C 180,E1 -19361.957,E2 -19361.957} C_VEL
LIN {X 0,Y 242.317,Z 257.497,A -85,B 0,C 180,E1 -19363.416,E2 -19363.416} C_VEL
LIN {X 0,Y 242.177,Z 256.859,A -85,B 0,C 180,E1 -19363.851,E2 -19363.851} C_VEL
LIN {X 0,Y 242.126,Z 256.821,A -85,B 0,C 180,E1 -19366.873,E2 -19366.873} C_VEL
LIN {X 0,Y 242.051,Z 256.829,A -85,B 0,C 180,E1 -19371.728,E2 -19371.728} C_VEL
LIN {X 0,Y 242.029,Z 256.793,A -85,B 0,C 180,E1 -19375.842,E2 -19375.842} C_VEL
LIN {X 0,Y 242.054,Z 256.815,A -85,B 0,C 180,E1 -19379.576,E2 -19379.576} C_VEL
LIN {X 0,Y 241.982,Z 256.837,A -85,B 0,C 180,E1 -19383.491,E2 -19383.491} C_VEL
LIN {X 0,Y 242.004,Z 256.837,A -85,B 0,C 180,E1 -19387.578,E2 -19387.578} C_VEL
LIN {X 0,Y 242.022,Z 256.813,A -85,B 0,C 180,E1 -19391.903,E2 -19391.903} C_VEL
LIN {X 0,Y 241.997,Z 256.84,A -85,B 0,C 180,E1 -19396.555,E2 -19396.555} C_VEL
LIN {X 0,Y 241.984,Z 256.813,A -85,B 0,C 180,E1 -19400.298,E2 -19400.298} C_VEL
LIN {X 0,Y 242.013,Z 256.83,A -85,B 0,C 180,E1 -19404.505,E2 -19404.505} C_VEL
LIN {X 0,Y 241.954,Z 256.838,A -85,B 0,C 180,E1 -19408.487,E2 -19408.487} C_VEL
LIN {X 0,Y 241.989,Z 256.798,A -85,B 0,C 180,E1 -19412.32,E2 -19412.32} C_VEL
LIN {X 0,Y 242.045,Z 256.825,A -85,B 0,C 180,E1 -19416.024,E2 -19416.024} C_VEL
LIN {X 0,Y 242.058,Z 256.829,A -85,B 0,C 180,E1 -19419.619,E2 -19419.619} C_VEL
LIN {X 0,Y 242.151,Z 256.782,A -85,B 0,C 180,E1 -19423.286,E2 -19423.286} C_VEL
LIN {X 0,Y 242.177,Z 256.804,A -85,B 0,C 180,E1 -19428.288,E2 -19428.288} C_VEL
LIN {X 0,Y 242.428,Z 256.786,A -85,B 0,C 180,E1 -19431.674,E2 -19431.674} C_VEL
LIN {X 0,Y 242.254,Z 256.784,A -85,B 0,C 180,E1 -19435.015,E2 -19435.015} C_VEL
LIN {X 0,Y 242.632,Z 256.713,A -85,B 0,C 180,E1 -19438.348,E2 -19438.348} C_VEL
LIN {X 0,Y 242.633,Z 256.749,A -85,B 0,C 180,E1 -19441.667,E2 -19441.667} C_VEL
LIN {X 0,Y 242.4,Z 256.779,A -85,B 0,C 180,E1 -19446.701,E2 -19446.701} C_VEL
LIN {X 0,Y 242.269,Z 256.764,A -85,B 0,C 180,E1 -19450.031,E2 -19450.031} C_VEL
LIN {X 0,Y 242.145,Z 256.811,A -85,B 0,C 180,E1 -19453.911,E2 -19453.911} C_VEL
LIN {X 0,Y 241.459,Z 256.907,A -85,B 0,C 180,E1 -19455.298,E2 -19455.298} C_VEL
LIN {X 0,Y 238.593,Z 257.261,A -85,B 0,C 180,E1 -19457.56,E2 -19457.56} C_VEL
LIN {X 0,Y 236.153,Z 257.546,A -85,B 0,C 180,E1 -19459.402,E2 -19459.402} C_VEL
LIN {X 0,Y 235.089,Z 257.668,A -85,B 0,C 180,E1 -19460.833,E2 -19460.833} C_VEL
LIN {X 0,Y 234.992,Z 257.68,A -85,B 0,C 180,E1 -19461.318,E2 -19461.318} C_VEL
LIN {X 0,Y 235.002,Z 257.714,A -85,B 0,C 180,E1 -19466.212,E2 -19466.212} C_VEL
LIN {X 0,Y 234.912,Z 257.701,A -85,B 0,C 180,E1 -19470.578,E2 -19470.578} C_VEL
LIN {X 0,Y 234.936,Z 257.723,A -85,B 0,C 180,E1 -19474.644,E2 -19474.644} C_VEL
LIN {X 0,Y 234.955,Z 257.712,A -85,B 0,C 180,E1 -19478.95,E2 -19478.95} C_VEL
LIN {X 0,Y 234.889,Z 257.688,A -85,B 0,C 180,E1 -19483.494,E2 -19483.494} C_VEL
LIN {X 0,Y 234.869,Z 257.687,A -85,B 0,C 180,E1 -19486.511,E2 -19486.511} C_VEL
LIN {X 0,Y 234.934,Z 257.708,A -85,B 0,C 180,E1 -19491.083,E2 -19491.083} C_VEL
LIN {X 0,Y 235.011,Z 257.822,A -85,B 0,C 180,E1 -19495.562,E2 -19495.562} C_VEL
LIN {X 0,Y 236.886,Z 266.679,A -85,B 0,C 180,E1 -19499.303,E2 -19499.303} C_VEL
LIN {X 0,Y 238.225,Z 270.452,A -85,B 0,C 180,E1 -19499.689,E2 -19499.689} C_VEL
LIN {X 0,Y 244.403,Z 287.677,A -85,B 0,C 180,E1 -19500.891,E2 -19500.891} C_VEL
LIN {X 0,Y 247.83,Z 312.954,A -85,B 0,C 180,E1 -19502.023,E2 -19502.023} C_VEL
LIN {X 0,Y 245.913,Z 374.58,A -85,B 0,C 180,E1 -19503.821,E2 -19503.821} C_VEL
LIN {X 0,Y 244.982,Z 387.099,A -85,B 0,C 180,E1 -19504.456,E2 -19504.456} C_VEL
LIN {X 0,Y 243.776,Z 399.533,A -85,B 0,C 180,E1 -19505.404,E2 -19505.404} C_VEL
LIN {X 0,Y 242.159,Z 412.027,A -85,B 0,C 180,E1 -19506.708,E2 -19506.708} C_VEL
LIN {X 0,Y 240.33,Z 423.751,A -85,B 0,C 180,E1 -19508.335,E2 -19508.335} C_VEL
LIN {X 0,Y 238.753,Z 434.331,A -85,B 0,C 180,E1 -19510.215,E2 -19510.215} C_VEL
LIN {X 0,Y 237.202,Z 443.803,A -85,B 0,C 180,E1 -19512.321,E2 -19512.321} C_VEL
LIN {X 0,Y 235.797,Z 451.551,A -85,B 0,C 180,E1 -19514.441,E2 -19514.441} C_VEL
LIN {X 0,Y 234.426,Z 459.119,A -85,B 0,C 180,E1 -19517.007,E2 -19517.007} C_VEL
LIN {X 0,Y 233.584,Z 465.196,A -85,B 0,C 180,E1 -19519.6,E2 -19519.6} C_VEL
LIN {X 0,Y 233.018,Z 469.98,A -85,B 0,C 180,E1 -19522.2,E2 -19522.2} C_VEL
LIN {X 0,Y 232.709,Z 473.621,A -85,B 0,C 180,E1 -19524.802,E2 -19524.802} C_VEL
LIN {X 0,Y 232.659,Z 475.495,A -85,B 0,C 180,E1 -19526.537,E2 -19526.537} C_VEL
LIN {X 0,Y 232.681,Z 476.895,A -85,B 0,C 180,E1 -19528.27,E2 -19528.27} C_VEL
LIN {X 0,Y 232.731,Z 477.886,A -85,B 0,C 180,E1 -19530.001,E2 -19530.001} C_VEL
LIN {X 0,Y 232.681,Z 478.484,A -85,B 0,C 180,E1 -19531.731,E2 -19531.731} C_VEL
LIN {X 0,Y 232.758,Z 478.574,A -85,B 0,C 180,E1 -19534.791,E2 -19534.791} C_VEL
LIN {X 0,Y 233.003,Z 477.88,A -85,B 0,C 180,E1 -19536.93,E2 -19536.93} C_VEL
LIN {X 0,Y 233.883,Z 475.529,A -85,B 0,C 180,E1 -19540.387,E2 -19540.387} C_VEL
LIN {X 0,Y 235.029,Z 472.652,A -85,B 0,C 180,E1 -19542.96,E2 -19542.96} C_VEL
LIN {X 0,Y 236.507,Z 468.776,A -85,B 0,C 180,E1 -19545.513,E2 -19545.513} C_VEL
LIN {X 0,Y 238.628,Z 463.793,A -85,B 0,C 180,E1 -19548.014,E2 -19548.014} C_VEL
LIN {X 0,Y 241.098,Z 457.561,A -85,B 0,C 180,E1 -19550.476,E2 -19550.476} C_VEL
LIN {X 0,Y 243.674,Z 450.111,A -85,B 0,C 180,E1 -19552.826,E2 -19552.826} C_VEL
LIN {X 0,Y 246.537,Z 441.938,A -85,B 0,C 180,E1 -19554.865,E2 -19554.865} C_VEL
LIN {X 0,Y 249.654,Z 432.344,A -85,B 0,C 180,E1 -19556.771,E2 -19556.771} C_VEL
LIN {X 0,Y 252.673,Z 421.721,A -85,B 0,C 180,E1 -19558.446,E2 -19558.446} C_VEL
LIN {X 0,Y 255.195,Z 411.442,A -85,B 0,C 180,E1 -19559.717,E2 -19559.717} C_VEL
LIN {X 0,Y 257.638,Z 399.163,A -85,B 0,C 180,E1 -19560.876,E2 -19560.876} C_VEL
LIN {X 0,Y 259.616,Z 386.31,A -85,B 0,C 180,E1 -19561.749,E2 -19561.749} C_VEL
LIN {X 0,Y 260.897,Z 373.892,A -85,B 0,C 180,E1 -19562.314,E2 -19562.314} C_VEL
LIN {X 0,Y 263.508,Z 319.026,A -85,B 0,C 180,E1 -19563.835,E2 -19563.835} C_VEL
LIN {X 0,Y 262.175,Z 311.989,A -85,B 0,C 180,E1 -19564.333,E2 -19564.333} C_VEL
LIN {X 0,Y 256.382,Z 299.235,A -85,B 0,C 180,E1 -19565.928,E2 -19565.928} C_VEL
LIN {X 0,Y 249.168,Z 285.288,A -85,B 0,C 180,E1 -19567.997,E2 -19567.997} C_VEL
LIN {X 0,Y 243.452,Z 275.699,A -85,B 0,C 180,E1 -19569.742,E2 -19569.742} C_VEL
LIN {X 0,Y 239.817,Z 270.125,A -85,B 0,C 180,E1 -19570.906,E2 -19570.906} C_VEL
LIN {X 0,Y 237.331,Z 265.877,A -85,B 0,C 180,E1 -19571.869,E2 -19571.869} C_VEL
LIN {X 0,Y 235.645,Z 260.214,A -85,B 0,C 180,E1 -19575.258,E2 -19575.258} C_VEL
LIN {X 0,Y 234.883,Z 257.731,A -85,B 0,C 180,E1 -19577.089,E2 -19577.089} C_VEL
LIN {X 0,Y 234.934,Z 257.715,A -85,B 0,C 180,E1 -19581.074,E2 -19581.074} C_VEL
LIN {X 0,Y 234.94,Z 257.715,A -85,B 0,C 180,E1 -19585.356,E2 -19585.356} C_VEL
LIN {X 0,Y 234.912,Z 257.722,A -85,B 0,C 180,E1 -19589.422,E2 -19589.422} C_VEL
LIN {X 0,Y 234.953,Z 257.719,A -85,B 0,C 180,E1 -19593.815,E2 -19593.815} C_VEL
LIN {X 0,Y 234.95,Z 257.711,A -85,B 0,C 180,E1 -19598.957,E2 -19598.957} C_VEL
LIN {X 0,Y 235.066,Z 257.699,A -85,B 0,C 180,E1 -19603.086,E2 -19603.086} C_VEL
LIN {X 0,Y 235.112,Z 257.691,A -85,B 0,C 180,E1 -19607.915,E2 -19607.915} C_VEL
LIN {X 0,Y 235.328,Z 257.672,A -85,B 0,C 180,E1 -19611.405,E2 -19611.405} C_VEL
LIN {X 0,Y 235.363,Z 257.655,A -85,B 0,C 180,E1 -19613.133,E2 -19613.133} C_VEL
LIN {X 0,Y 235.584,Z 257.626,A -85,B 0,C 180,E1 -19618.283,E2 -19618.283} C_VEL
LIN {X 0,Y 235.591,Z 257.633,A -85,B 0,C 180,E1 -19621.702,E2 -19621.702} C_VEL
LIN {X 0,Y 235.35,Z 257.657,A -85,B 0,C 180,E1 -19626.852,E2 -19626.852} C_VEL
LIN {X 0,Y 235.21,Z 257.68,A -85,B 0,C 180,E1 -19630.319,E2 -19630.319} C_VEL
LIN {X 0,Y 235.086,Z 257.692,A -85,B 0,C 180,E1 -19635.6,E2 -19635.6} C_VEL
LIN {X 0,Y 234.99,Z 257.706,A -85,B 0,C 180,E1 -19639.198,E2 -19639.198} C_VEL
LIN {X 0,Y 234.949,Z 257.715,A -85,B 0,C 180,E1 -19642.875,E2 -19642.875} C_VEL
LIN {X 0,Y 234.97,Z 257.788,A -85,B 0,C 180,E1 -19647.369,E2 -19647.369} C_VEL
LIN {X 0,Y 236.125,Z 261.597,A -85,B 0,C 180,E1 -19649.854,E2 -19649.854} C_VEL
LIN {X 0,Y 238.915,Z 266.081,A -85,B 0,C 180,E1 -19650.911,E2 -19650.911} C_VEL
LIN {X 0,Y 243.745,Z 273.319,A -85,B 0,C 180,E1 -19652.463,E2 -19652.463} C_VEL
LIN {X 0,Y 249.652,Z 283.053,A -85,B 0,C 180,E1 -19654.255,E2 -19654.255} C_VEL
LIN {X 0,Y 255.907,Z 294.367,A -85,B 0,C 180,E1 -19656.026,E2 -19656.026} C_VEL
LIN {X 0,Y 262.368,Z 308.01,A -85,B 0,C 180,E1 -19657.793,E2 -19657.793} C_VEL
LIN {X 0,Y 263.907,Z 311.806,A -85,B 0,C 180,E1 -19658.214,E2 -19658.214} C_VEL
LIN {X 0,Y 261.077,Z 368.843,A -85,B 0,C 180,E1 -19659.785,E2 -19659.785} C_VEL
LIN {X 0,Y 259.726,Z 381.426,A -85,B 0,C 180,E1 -19660.371,E2 -19660.371} C_VEL
LIN {X 0,Y 257.829,Z 394.399,A -85,B 0,C 180,E1 -19661.296,E2 -19661.296} C_VEL
LIN {X 0,Y 255.615,Z 405.506,A -85,B 0,C 180,E1 -19662.361,E2 -19662.361} C_VEL
LIN {X 0,Y 252.947,Z 416.536,A -85,B 0,C 180,E1 -19663.747,E2 -19663.747} C_VEL
LIN {X 0,Y 249.809,Z 427.837,A -85,B 0,C 180,E1 -19665.587,E2 -19665.587} C_VEL
LIN {X 0,Y 246.788,Z 437.341,A -85,B 0,C 180,E1 -19667.556,E2 -19667.556} C_VEL
LIN {X 0,Y 244.016,Z 445.223,A -85,B 0,C 180,E1 -19669.606,E2 -19669.606} C_VEL
LIN {X 0,Y 240.99,Z 453.199,A -85,B 0,C 180,E1 -19672.235,E2 -19672.235} C_VEL
LIN {X 0,Y 238.399,Z 459.515,A -85,B 0,C 180,E1 -19674.91,E2 -19674.91} C_VEL
LIN {X 0,Y 236.341,Z 464.395,A -85,B 0,C 180,E1 -19677.638,E2 -19677.638} C_VEL
LIN {X 0,Y 234.889,Z 467.766,A -85,B 0,C 180,E1 -19680.171,E2 -19680.171} C_VEL
LIN {X 0,Y 233.644,Z 470.488,A -85,B 0,C 180,E1 -19683.179,E2 -19683.179} C_VEL
LIN {X 0,Y 233.149,Z 471.536,A -85,B 0,C 180,E1 -19685.038,E2 -19685.038} C_VEL
LIN {X 0,Y 232.718,Z 472.155,A -85,B 0,C 180,E1 -19686.883,E2 -19686.883} C_VEL
LIN {X 0,Y 232.413,Z 472.226,A -85,B 0,C 180,E1 -19689.593,E2 -19689.593} C_VEL
LIN {X 0,Y 232.263,Z 471.3,A -85,B 0,C 180,E1 -19692.386,E2 -19692.386} C_VEL
LIN {X 0,Y 232.454,Z 469.22,A -85,B 0,C 180,E1 -19695.308,E2 -19695.308} C_VEL
LIN {X 0,Y 232.792,Z 466.47,A -85,B 0,C 180,E1 -19697.799,E2 -19697.799} C_VEL
LIN {X 0,Y 233.238,Z 462.488,A -85,B 0,C 180,E1 -19700.46,E2 -19700.46} C_VEL
LIN {X 0,Y 234.004,Z 457.328,A -85,B 0,C 180,E1 -19703.1,E2 -19703.1} C_VEL
LIN {X 0,Y 235.066,Z 450.819,A -85,B 0,C 180,E1 -19705.713,E2 -19705.713} C_VEL
LIN {X 0,Y 236.409,Z 442.681,A -85,B 0,C 180,E1 -19708.296,E2 -19708.296} C_VEL
LIN {X 0,Y 237.839,Z 434.37,A -85,B 0,C 180,E1 -19710.423,E2 -19710.423} C_VEL
LIN {X 0,Y 239.544,Z 424.624,A -85,B 0,C 180,E1 -19712.44,E2 -19712.44} C_VEL
LIN {X 0,Y 241.237,Z 414.064,A -85,B 0,C 180,E1 -19714.176,E2 -19714.176} C_VEL
LIN {X 0,Y 242.764,Z 403.052,A -85,B 0,C 180,E1 -19715.607,E2 -19715.607} C_VEL
LIN {X 0,Y 244.109,Z 390.922,A -85,B 0,C 180,E1 -19716.82,E2 -19716.82} C_VEL
LIN {X 0,Y 245.209,Z 378.411,A -85,B 0,C 180,E1 -19717.72,E2 -19717.72} C_VEL
LIN {X 0,Y 245.978,Z 365.206,A -85,B 0,C 180,E1 -19718.324,E2 -19718.324} C_VEL
LIN {X 0,Y 248.077,Z 300.888,A -85,B 0,C 180,E1 -19720.17,E2 -19720.17} C_VEL
LIN {X 0,Y 246.172,Z 289.43,A -85,B 0,C 180,E1 -19720.718,E2 -19720.718} C_VEL
LIN {X 0,Y 241.326,Z 275,A -85,B 0,C 180,E1 -19721.675,E2 -19721.675} C_VEL
LIN {X 0,Y 235.985,Z 261.528,A -85,B 0,C 180,E1 -19722.716,E2 -19722.716} C_VEL
LIN {X 0,Y 235.767,Z 260.693,A -85,B 0,C 180,E1 -19722.919,E2 -19722.919} C_VEL
LIN {X 0,Y 235.121,Z 257.766,A -85,B 0,C 180,E1 -19724.276,E2 -19724.276} C_VEL
LIN {X 0,Y 235.063,Z 257.689,A -85,B 0,C 180,E1 -19727.396,E2 -19727.396} C_VEL
LIN {X 0,Y 235.012,Z 257.71,A -85,B 0,C 180,E1 -19732.048,E2 -19732.048} C_VEL
LIN {X 0,Y 234.938,Z 257.671,A -85,B 0,C 180,E1 -19736.66,E2 -19736.66} C_VEL
LIN {X 0,Y 234.943,Z 257.716,A -85,B 0,C 180,E1 -19740.565,E2 -19740.565} C_VEL
LIN {X 0,Y 234.948,Z 257.704,A -85,B 0,C 180,E1 -19744.634,E2 -19744.634} C_VEL
LIN {X 0,Y 234.965,Z 257.717,A -85,B 0,C 180,E1 -19748.967,E2 -19748.967} C_VEL
LIN {X 0,Y 234.969,Z 257.695,A -85,B 0,C 180,E1 -19753.466,E2 -19753.466} C_VEL
LIN {X 0,Y 234.969,Z 257.716,A -85,B 0,C 180,E1 -19756.546,E2 -19756.546} C_VEL
LIN {X 0,Y 234.929,Z 257.686,A -85,B 0,C 180,E1 -19761.093,E2 -19761.093} C_VEL
LIN {X 0,Y 234.937,Z 257.717,A -85,B 0,C 180,E1 -19765.374,E2 -19765.374} C_VEL
LIN {X 0,Y 234.949,Z 257.692,A -85,B 0,C 180,E1 -19770.165,E2 -19770.165} C_VEL
LIN {X 0,Y 234.976,Z 257.68,A -85,B 0,C 180,E1 -19773.801,E2 -19773.801} C_VEL
LIN {X 0,Y 235.027,Z 257.708,A -85,B 0,C 180,E1 -19778.981,E2 -19778.981} C_VEL
LIN {X 0,Y 235.104,Z 257.661,A -85,B 0,C 180,E1 -19783.051,E2 -19783.051} C_VEL
LIN {X 0,Y 235.109,Z 257.678,A -85,B 0,C 180,E1 -19787.93,E2 -19787.93} C_VEL
LIN {X 0,Y 235.383,Z 257.665,A -85,B 0,C 180,E1 -19791.422,E2 -19791.422} C_VEL
LIN {X 0,Y 235.399,Z 257.656,A -85,B 0,C 180,E1 -19793.149,E2 -19793.149} C_VEL
LIN {X 0,Y 235.592,Z 257.589,A -85,B 0,C 180,E1 -19798.298,E2 -19798.298} C_VEL
LIN {X 0,Y 235.593,Z 257.626,A -85,B 0,C 180,E1 -19801.717,E2 -19801.717} C_VEL
LIN {X 0,Y 235.353,Z 257.657,A -85,B 0,C 180,E1 -19806.868,E2 -19806.868} C_VEL
LIN {X 0,Y 235.216,Z 257.642,A -85,B 0,C 180,E1 -19810.335,E2 -19810.335} C_VEL
LIN {X 0,Y 235.119,Z 257.696,A -85,B 0,C 180,E1 -19815.613,E2 -19815.613} C_VEL
LIN {X 0,Y 235.013,Z 257.69,A -85,B 0,C 180,E1 -19819.212,E2 -19819.212} C_VEL
LIN {X 0,Y 234.992,Z 257.68,A -85,B 0,C 180,E1 -19821.318,E2 -19821.318} C_VEL
LIN {X 0,Y 234.281,Z 257.781,A -85,B 0,C 180,E1 -19822.749,E2 -19822.749} C_VEL
LIN {X 0,Y 231.37,Z 258.167,A -85,B 0,C 180,E1 -19825.082,E2 -19825.082} C_VEL
LIN {X 0,Y 228.937,Z 258.465,A -85,B 0,C 180,E1 -19826.985,E2 -19826.985} C_VEL
LIN {X 0,Y 227.925,Z 258.577,A -85,B 0,C 180,E1 -19828.464,E2 -19828.464} C_VEL
LIN {X 0,Y 227.859,Z 258.579,A -85,B 0,C 180,E1 -19828.965,E2 -19828.965} C_VEL
LIN {X 0,Y 227.888,Z 258.602,A -85,B 0,C 180,E1 -19833.726,E2 -19833.726} C_VEL
LIN {X 0,Y 227.852,Z 258.59,A -85,B 0,C 180,E1 -19838.097,E2 -19838.097} C_VEL
LIN {X 0,Y 227.818,Z 258.58,A -85,B 0,C 180,E1 -19842.749,E2 -19842.749} C_VEL
LIN {X 0,Y 227.831,Z 258.554,A -85,B 0,C 180,E1 -19845.202,E2 -19845.202} C_VEL
LIN {X 0,Y 227.813,Z 258.609,A -85,B 0,C 180,E1 -19849.621,E2 -19849.621} C_VEL
LIN {X 0,Y 227.888,Z 258.601,A -85,B 0,C 180,E1 -19854.13,E2 -19854.13} C_VEL
LIN {X 0,Y 227.97,Z 258.816,A -85,B 0,C 180,E1 -19855.094,E2 -19855.094} C_VEL
LIN {X 0,Y 229.644,Z 266.695,A -85,B 0,C 180,E1 -19858.494,E2 -19858.494} C_VEL
LIN {X 0,Y 231.45,Z 271.458,A -85,B 0,C 180,E1 -19858.965,E2 -19858.965} C_VEL
LIN {X 0,Y 238.095,Z 289.837,A -85,B 0,C 180,E1 -19860.314,E2 -19860.314} C_VEL
LIN {X 0,Y 241.224,Z 314.26,A -85,B 0,C 180,E1 -19861.429,E2 -19861.429} C_VEL
LIN {X 0,Y 239.225,Z 375.358,A -85,B 0,C 180,E1 -19863.266,E2 -19863.266} C_VEL
LIN {X 0,Y 238.205,Z 388.355,A -85,B 0,C 180,E1 -19863.969,E2 -19863.969} C_VEL
LIN {X 0,Y 236.921,Z 401.012,A -85,B 0,C 180,E1 -19864.995,E2 -19864.995} C_VEL
LIN {X 0,Y 235.366,Z 412.238,A -85,B 0,C 180,E1 -19866.228,E2 -19866.228} C_VEL
LIN {X 0,Y 233.481,Z 423.905,A -85,B 0,C 180,E1 -19867.898,E2 -19867.898} C_VEL
LIN {X 0,Y 231.755,Z 434.851,A -85,B 0,C 180,E1 -19869.912,E2 -19869.912} C_VEL
LIN {X 0,Y 230.065,Z 444.686,A -85,B 0,C 180,E1 -19872.214,E2 -19872.214} C_VEL
LIN {X 0,Y 228.367,Z 453.638,A -85,B 0,C 180,E1 -19874.836,E2 -19874.836} C_VEL
LIN {X 0,Y 227.133,Z 460.8,A -85,B 0,C 180,E1 -19877.492,E2 -19877.492} C_VEL
LIN {X 0,Y 226.34,Z 466.496,A -85,B 0,C 180,E1 -19880.168,E2 -19880.168} C_VEL
LIN {X 0,Y 225.838,Z 470.96,A -85,B 0,C 180,E1 -19882.85,E2 -19882.85} C_VEL
LIN {X 0,Y 225.602,Z 474.323,A -85,B 0,C 180,E1 -19885.535,E2 -19885.535} C_VEL
LIN {X 0,Y 225.581,Z 476.682,A -85,B 0,C 180,E1 -19888.215,E2 -19888.215} C_VEL
LIN {X 0,Y 225.647,Z 477.707,A -85,B 0,C 180,E1 -19890.001,E2 -19890.001} C_VEL
LIN {X 0,Y 225.581,Z 478.336,A -85,B 0,C 180,E1 -19891.786,E2 -19891.786} C_VEL
LIN {X 0,Y 225.659,Z 478.52,A -85,B 0,C 180,E1 -19894.646,E2 -19894.646} C_VEL
LIN {X 0,Y 225.946,Z 477.861,A -85,B 0,C 180,E1 -19897.148,E2 -19897.148} C_VEL
LIN {X 0,Y 226.889,Z 475.575,A -85,B 0,C 180,E1 -19900.711,E2 -19900.711} C_VEL
LIN {X 0,Y 228.099,Z 472.768,A -85,B 0,C 180,E1 -19903.361,E2 -19903.361} C_VEL
LIN {X 0,Y 229.664,Z 468.972,A -85,B 0,C 180,E1 -19905.987,E2 -19905.987} C_VEL
LIN {X 0,Y 231.883,Z 464.077,A -85,B 0,C 180,E1 -19908.557,E2 -19908.557} C_VEL
LIN {X 0,Y 234.456,Z 457.947,A -85,B 0,C 180,E1 -19911.083,E2 -19911.083} C_VEL
LIN {X 0,Y 237.296,Z 450.358,A -85,B 0,C 180,E1 -19913.568,E2 -19913.568} C_VEL
LIN {X 0,Y 240.774,Z 440.845,A -85,B 0,C 180,E1 -19915.966,E2 -19915.966} C_VEL
LIN {X 0,Y 244.06,Z 431.052,A -85,B 0,C 180,E1 -19917.901,E2 -19917.901} C_VEL
LIN {X 0,Y 247.209,Z 420.099,A -85,B 0,C 180,E1 -19919.602,E2 -19919.602} C_VEL
LIN {X 0,Y 249.872,Z 409.401,A -85,B 0,C 180,E1 -19920.885,E2 -19920.885} C_VEL
LIN {X 0,Y 252.451,Z 396.551,A -85,B 0,C 180,E1 -19922.052,E2 -19922.052} C_VEL
LIN {X 0,Y 254.33,Z 384.216,A -85,B 0,C 180,E1 -19922.841,E2 -19922.841} C_VEL
LIN {X 0,Y 255.587,Z 370.225,A -85,B 0,C 180,E1 -19923.423,E2 -19923.423} C_VEL
LIN {X 0,Y 258.039,Z 320.244,A -85,B 0,C 180,E1 -19924.813,E2 -19924.813} C_VEL
LIN {X 0,Y 256.951,Z 314.856,A -85,B 0,C 180,E1 -19925.226,E2 -19925.226} C_VEL
LIN {X 0,Y 251.029,Z 301.736,A -85,B 0,C 180,E1 -19926.94,E2 -19926.94} C_VEL
LIN {X 0,Y 244.33,Z 288.939,A -85,B 0,C 180,E1 -19928.963,E2 -19928.963} C_VEL
LIN {X 0,Y 239.621,Z 280.855,A -85,B 0,C 180,E1 -19930.478,E2 -19930.478} C_VEL
LIN {X 0,Y 235.949,Z 275.119,A -85,B 0,C 180,E1 -19931.71,E2 -19931.71} C_VEL
LIN {X 0,Y 232.696,Z 270.123,A -85,B 0,C 180,E1 -19932.857,E2 -19932.857} C_VEL
LIN {X 0,Y 230.067,Z 265.738,A -85,B 0,C 180,E1 -19933.956,E2 -19933.956} C_VEL
LIN {X 0,Y 228.226,Z 260.172,A -85,B 0,C 180,E1 -19937.652,E2 -19937.652} C_VEL
LIN {X 0,Y 227.839,Z 258.607,A -85,B 0,C 180,E1 -19938.983,E2 -19938.983} C_VEL
LIN {X 0,Y 227.895,Z 258.598,A -85,B 0,C 180,E1 -19943.304,E2 -19943.304} C_VEL
LIN {X 0,Y 227.894,Z 258.6,A -85,B 0,C 180,E1 -19946.373,E2 -19946.373} C_VEL
LIN {X 0,Y 227.888,Z 258.595,A -85,B 0,C 180,E1 -19950.426,E2 -19950.426} C_VEL
LIN {X 0,Y 227.878,Z 258.595,A -85,B 0,C 180,E1 -19954.412,E2 -19954.412} C_VEL
LIN {X 0,Y 227.931,Z 258.593,A -85,B 0,C 180,E1 -19958.277,E2 -19958.277} C_VEL
LIN {X 0,Y 228.03,Z 258.567,A -85,B 0,C 180,E1 -19963.888,E2 -19963.888} C_VEL
LIN {X 0,Y 228.069,Z 258.572,A -85,B 0,C 180,E1 -19967.535,E2 -19967.535} C_VEL
LIN {X 0,Y 228.266,Z 258.551,A -85,B 0,C 180,E1 -19971.137,E2 -19971.137} C_VEL
LIN {X 0,Y 228.316,Z 258.534,A -85,B 0,C 180,E1 -19972.92,E2 -19972.92} C_VEL
LIN {X 0,Y 228.542,Z 258.503,A -85,B 0,C 180,E1 -19978.23,E2 -19978.23} C_VEL
LIN {X 0,Y 228.549,Z 258.509,A -85,B 0,C 180,E1 -19981.754,E2 -19981.754} C_VEL
LIN {X 0,Y 228.302,Z 258.534,A -85,B 0,C 180,E1 -19987.065,E2 -19987.065} C_VEL
LIN {X 0,Y 228.141,Z 258.558,A -85,B 0,C 180,E1 -19990.643,E2 -19990.643} C_VEL
LIN {X 0,Y 228.044,Z 258.573,A -85,B 0,C 180,E1 -19994.265,E2 -19994.265} C_VEL
LIN {X 0,Y 227.989,Z 258.58,A -85,B 0,C 180,E1 -19997.945,E2 -19997.945} C_VEL
LIN {X 0,Y 227.918,Z 258.587,A -85,B 0,C 180,E1 -20002.321,E2 -20002.321} C_VEL
LIN {X 0,Y 227.932,Z 258.686,A -85,B 0,C 180,E1 -20005.564,E2 -20005.564} C_VEL
LIN {X 0,Y 228.956,Z 261.887,A -85,B 0,C 180,E1 -20007.777,E2 -20007.777} C_VEL
LIN {X 0,Y 231.84,Z 266.281,A -85,B 0,C 180,E1 -20008.942,E2 -20008.942} C_VEL
LIN {X 0,Y 237.127,Z 274.187,A -85,B 0,C 180,E1 -20010.799,E2 -20010.799} C_VEL
LIN {X 0,Y 240.098,Z 278.773,A -85,B 0,C 180,E1 -20011.785,E2 -20011.785} C_VEL
LIN {X 0,Y 246.553,Z 289.595,A -85,B 0,C 180,E1 -20013.82,E2 -20013.82} C_VEL
LIN {X 0,Y 253.219,Z 302.303,A -85,B 0,C 180,E1 -20015.778,E2 -20015.778} C_VEL
LIN {X 0,Y 258.342,Z 313.78,A -85,B 0,C 180,E1 -20017.239,E2 -20017.239} C_VEL
LIN {X 0,Y 255.457,Z 369.774,A -85,B 0,C 180,E1 -20018.826,E2 -20018.826} C_VEL
LIN {X 0,Y 253.918,Z 383.211,A -85,B 0,C 180,E1 -20019.488,E2 -20019.488} C_VEL
LIN {X 0,Y 252.094,Z 394.967,A -85,B 0,C 180,E1 -20020.363,E2 -20020.363} C_VEL
LIN {X 0,Y 249.747,Z 406.204,A -85,B 0,C 180,E1 -20021.475,E2 -20021.475} C_VEL
LIN {X 0,Y 246.897,Z 417.379,A -85,B 0,C 180,E1 -20022.922,E2 -20022.922} C_VEL
LIN {X 0,Y 243.719,Z 428.329,A -85,B 0,C 180,E1 -20024.757,E2 -20024.757} C_VEL
LIN {X 0,Y 240.421,Z 438.086,A -85,B 0,C 180,E1 -20026.846,E2 -20026.846} C_VEL
LIN {X 0,Y 237.06,Z 447.009,A -85,B 0,C 180,E1 -20029.29,E2 -20029.29} C_VEL
LIN {X 0,Y 233.965,Z 454.666,A -85,B 0,C 180,E1 -20031.99,E2 -20031.99} C_VEL
LIN {X 0,Y 231.344,Z 460.639,A -85,B 0,C 180,E1 -20034.746,E2 -20034.746} C_VEL
LIN {X 0,Y 229.229,Z 465.252,A -85,B 0,C 180,E1 -20037.551,E2 -20037.551} C_VEL
LIN {X 0,Y 227.637,Z 468.647,A -85,B 0,C 180,E1 -20040.397,E2 -20040.397} C_VEL
LIN {X 0,Y 226.829,Z 470.304,A -85,B 0,C 180,E1 -20042.305,E2 -20042.305} C_VEL
LIN {X 0,Y 226.205,Z 471.476,A -85,B 0,C 180,E1 -20044.267,E2 -20044.267} C_VEL
LIN {X 0,Y 225.77,Z 472.148,A -85,B 0,C 180,E1 -20046.129,E2 -20046.129} C_VEL
LIN {X 0,Y 225.356,Z 472.33,A -85,B 0,C 180,E1 -20049.293,E2 -20049.293} C_VEL
LIN {X 0,Y 225.163,Z 471.583,A -85,B 0,C 180,E1 -20051.812,E2 -20051.812} C_VEL
LIN {X 0,Y 225.332,Z 469.37,A -85,B 0,C 180,E1 -20055.17,E2 -20055.17} C_VEL
LIN {X 0,Y 225.767,Z 465.907,A -85,B 0,C 180,E1 -20058.326,E2 -20058.326} C_VEL
LIN {X 0,Y 226.275,Z 461.701,A -85,B 0,C 180,E1 -20061.065,E2 -20061.065} C_VEL
LIN {X 0,Y 227.17,Z 456.273,A -85,B 0,C 180,E1 -20063.783,E2 -20063.783} C_VEL
LIN {X 0,Y 228.267,Z 449.482,A -85,B 0,C 180,E1 -20066.469,E2 -20066.469} C_VEL
LIN {X 0,Y 229.759,Z 441.045,A -85,B 0,C 180,E1 -20069.123,E2 -20069.123} C_VEL
LIN {X 0,Y 231.333,Z 432.334,A -85,B 0,C 180,E1 -20071.305,E2 -20071.305} C_VEL
LIN {X 0,Y 233.302,Z 421.541,A -85,B 0,C 180,E1 -20073.453,E2 -20073.453} C_VEL
LIN {X 0,Y 234.957,Z 410.849,A -85,B 0,C 180,E1 -20075.148,E2 -20075.148} C_VEL
LIN {X 0,Y 236.555,Z 398.919,A -85,B 0,C 180,E1 -20076.61,E2 -20076.61} C_VEL
LIN {X 0,Y 237.845,Z 386.532,A -85,B 0,C 180,E1 -20077.747,E2 -20077.747} C_VEL
LIN {X 0,Y 238.926,Z 373.899,A -85,B 0,C 180,E1 -20078.554,E2 -20078.554} C_VEL
LIN {X 0,Y 239.574,Z 359.167,A -85,B 0,C 180,E1 -20079.114,E2 -20079.114} C_VEL
LIN {X 0,Y 241.497,Z 301.451,A -85,B 0,C 180,E1 -20080.799,E2 -20080.799} C_VEL
LIN {X 0,Y 239.821,Z 291.535,A -85,B 0,C 180,E1 -20081.291,E2 -20081.291} C_VEL
LIN {X 0,Y 235.118,Z 277.505,A -85,B 0,C 180,E1 -20082.256,E2 -20082.256} C_VEL
LIN {X 0,Y 228.76,Z 261.553,A -85,B 0,C 180,E1 -20083.567,E2 -20083.567} C_VEL
LIN {X 0,Y 228.29,Z 259.647,A -85,B 0,C 180,E1 -20084.257,E2 -20084.257} C_VEL
LIN {X 0,Y 228.083,Z 258.642,A -85,B 0,C 180,E1 -20084.84,E2 -20084.84} C_VEL
LIN {X 0,Y 227.987,Z 258.562,A -85,B 0,C 180,E1 -20087.954,E2 -20087.954} C_VEL
LIN {X 0,Y 227.944,Z 258.591,A -85,B 0,C 180,E1 -20092.364,E2 -20092.364} C_VEL
LIN {X 0,Y 227.909,Z 258.545,A -85,B 0,C 180,E1 -20096.608,E2 -20096.608} C_VEL
LIN {X 0,Y 227.922,Z 258.585,A -85,B 0,C 180,E1 -20100.322,E2 -20100.322} C_VEL
LIN {X 0,Y 227.92,Z 258.587,A -85,B 0,C 180,E1 -20103.712,E2 -20103.712} C_VEL
LIN {X 0,Y 227.867,Z 258.602,A -85,B 0,C 180,E1 -20108.086,E2 -20108.086} C_VEL
LIN {X 0,Y 227.911,Z 258.569,A -85,B 0,C 180,E1 -20112.718,E2 -20112.718} C_VEL
LIN {X 0,Y 227.906,Z 258.595,A -85,B 0,C 180,E1 -20117.293,E2 -20117.293} C_VEL
LIN {X 0,Y 227.846,Z 258.568,A -85,B 0,C 180,E1 -20121.921,E2 -20121.921} C_VEL
LIN {X 0,Y 227.868,Z 258.602,A -85,B 0,C 180,E1 -20126.38,E2 -20126.38} C_VEL
LIN {X 0,Y 227.899,Z 258.566,A -85,B 0,C 180,E1 -20130.446,E2 -20130.446} C_VEL
LIN {X 0,Y 227.912,Z 258.568,A -85,B 0,C 180,E1 -20134.434,E2 -20134.434} C_VEL
LIN {X 0,Y 227.99,Z 258.585,A -85,B 0,C 180,E1 -20138.299,E2 -20138.299} C_VEL
LIN {X 0,Y 228.033,Z 258.543,A -85,B 0,C 180,E1 -20142.825,E2 -20142.825} C_VEL
LIN {X 0,Y 228.065,Z 258.549,A -85,B 0,C 180,E1 -20147.552,E2 -20147.552} C_VEL
LIN {X 0,Y 228.318,Z 258.545,A -85,B 0,C 180,E1 -20151.155,E2 -20151.155} C_VEL
LIN {X 0,Y 228.352,Z 258.536,A -85,B 0,C 180,E1 -20152.937,E2 -20152.937} C_VEL
LIN {X 0,Y 228.55,Z 258.465,A -85,B 0,C 180,E1 -20158.246,E2 -20158.246} C_VEL
LIN {X 0,Y 228.551,Z 258.503,A -85,B 0,C 180,E1 -20161.77,E2 -20161.77} C_VEL
LIN {X 0,Y 228.305,Z 258.531,A -85,B 0,C 180,E1 -20167.081,E2 -20167.081} C_VEL
LIN {X 0,Y 228.147,Z 258.522,A -85,B 0,C 180,E1 -20170.659,E2 -20170.659} C_VEL
LIN {X 0,Y 228.067,Z 258.569,A -85,B 0,C 180,E1 -20174.279,E2 -20174.279} C_VEL
LIN {X 0,Y 228.009,Z 258.574,A -85,B 0,C 180,E1 -20177.96,E2 -20177.96} C_VEL
LIN {X 0,Y 227.924,Z 258.568,A -85,B 0,C 180,E1 -20182.327,E2 -20182.327} C_VEL
LIN {X 0,Y 227.949,Z 258.591,A -85,B 0,C 180,E1 -20186.607,E2 -20186.607} C_VEL
LIN {X 0,Y 227.859,Z 258.579,A -85,B 0,C 180,E1 -20188.965,E2 -20188.965} C_VEL
LIN {X 0,Y 227.566,Z 258.615,A -85,B 0,C 180,E1 -20189.952,E2 -20189.952} C_VEL
LIN {X 0,Y 226.216,Z 258.796,A -85,B 0,C 180,E1 -20191.409,E2 -20191.409} C_VEL
LIN {X 0,Y 221.862,Z 259.349,A -85,B 0,C 180,E1 -20194.813,E2 -20194.813} C_VEL
LIN {X 0,Y 220.862,Z 259.46,A -85,B 0,C 180,E1 -20196.341,E2 -20196.341} C_VEL
LIN {X 0,Y 220.81,Z 259.463,A -85,B 0,C 180,E1 -20196.858,E2 -20196.858} C_VEL
LIN {X 0,Y 220.808,Z 259.48,A -85,B 0,C 180,E1 -20200.193,E2 -20200.193} C_VEL
LIN {X 0,Y 220.776,Z 259.434,A -85,B 0,C 180,E1 -20204.462,E2 -20204.462} C_VEL
LIN {X 0,Y 220.761,Z 259.469,A -85,B 0,C 180,E1 -20208.047,E2 -20208.047} C_VEL
LIN {X 0,Y 220.842,Z 259.462,A -85,B 0,C 180,E1 -20212.797,E2 -20212.797} C_VEL
LIN {X 0,Y 220.915,Z 259.702,A -85,B 0,C 180,E1 -20214.509,E2 -20214.509} C_VEL
LIN {X 0,Y 222.435,Z 266.709,A -85,B 0,C 180,E1 -20217.637,E2 -20217.637} C_VEL
LIN {X 0,Y 226.782,Z 277.808,A -85,B 0,C 180,E1 -20218.638,E2 -20218.638} C_VEL
LIN {X 0,Y 231.763,Z 291.913,A -85,B 0,C 180,E1 -20219.699,E2 -20219.699} C_VEL
LIN {X 0,Y 234.667,Z 314.629,A -85,B 0,C 180,E1 -20220.776,E2 -20220.776} C_VEL
LIN {X 0,Y 232.67,Z 374.48,A -85,B 0,C 180,E1 -20222.607,E2 -20222.607} C_VEL
LIN {X 0,Y 231.662,Z 387.303,A -85,B 0,C 180,E1 -20223.297,E2 -20223.297} C_VEL
LIN {X 0,Y 230.298,Z 400.205,A -85,B 0,C 180,E1 -20224.345,E2 -20224.345} C_VEL
LIN {X 0,Y 228.588,Z 412.447,A -85,B 0,C 180,E1 -20225.719,E2 -20225.719} C_VEL
LIN {X 0,Y 226.646,Z 424.059,A -85,B 0,C 180,E1 -20227.436,E2 -20227.436} C_VEL
LIN {X 0,Y 224.936,Z 434.545,A -85,B 0,C 180,E1 -20229.422,E2 -20229.422} C_VEL
LIN {X 0,Y 223.565,Z 442.518,A -85,B 0,C 180,E1 -20231.288,E2 -20231.288} C_VEL
LIN {X 0,Y 222.059,Z 450.209,A -85,B 0,C 180,E1 -20233.451,E2 -20233.451} C_VEL
LIN {X 0,Y 220.544,Z 458.013,A -85,B 0,C 180,E1 -20236.173,E2 -20236.173} C_VEL
LIN {X 0,Y 219.582,Z 464.263,A -85,B 0,C 180,E1 -20238.929,E2 -20238.929} C_VEL
LIN {X 0,Y 218.914,Z 469.204,A -85,B 0,C 180,E1 -20241.694,E2 -20241.694} C_VEL
LIN {X 0,Y 218.58,Z 472.994,A -85,B 0,C 180,E1 -20244.465,E2 -20244.465} C_VEL
LIN {X 0,Y 218.47,Z 474.94,A -85,B 0,C 180,E1 -20246.312,E2 -20246.312} C_VEL
LIN {X 0,Y 218.483,Z 476.462,A -85,B 0,C 180,E1 -20248.157,E2 -20248.157} C_VEL
LIN {X 0,Y 218.565,Z 477.527,A -85,B 0,C 180,E1 -20250.001,E2 -20250.001} C_VEL
LIN {X 0,Y 218.484,Z 478.189,A -85,B 0,C 180,E1 -20251.844,E2 -20251.844} C_VEL
LIN {X 0,Y 218.653,Z 478.366,A -85,B 0,C 180,E1 -20255.534,E2 -20255.534} C_VEL
LIN {X 0,Y 219.318,Z 476.931,A -85,B 0,C 180,E1 -20259.22,E2 -20259.22} C_VEL
LIN {X 0,Y 220.701,Z 473.939,A -85,B 0,C 180,E1 -20262.88,E2 -20262.88} C_VEL
LIN {X 0,Y 222.245,Z 470.553,A -85,B 0,C 180,E1 -20265.593,E2 -20265.593} C_VEL
LIN {X 0,Y 224.347,Z 466.119,A -85,B 0,C 180,E1 -20268.257,E2 -20268.257} C_VEL
LIN {X 0,Y 227.437,Z 459.437,A -85,B 0,C 180,E1 -20271.29,E2 -20271.29} C_VEL
LIN {X 0,Y 230.257,Z 452.207,A -85,B 0,C 180,E1 -20273.855,E2 -20273.855} C_VEL
LIN {X 0,Y 233.802,Z 443.246,A -85,B 0,C 180,E1 -20276.32,E2 -20276.32} C_VEL
LIN {X 0,Y 237.535,Z 432.931,A -85,B 0,C 180,E1 -20278.496,E2 -20278.496} C_VEL
LIN {X 0,Y 240.773,Z 422.47,A -85,B 0,C 180,E1 -20280.233,E2 -20280.233} C_VEL
LIN {X 0,Y 243.886,Z 410.813,A -85,B 0,C 180,E1 -20281.73,E2 -20281.73} C_VEL
LIN {X 0,Y 246.555,Z 398.378,A -85,B 0,C 180,E1 -20282.914,E2 -20282.914} C_VEL
LIN {X 0,Y 248.683,Z 385.323,A -85,B 0,C 180,E1 -20283.807,E2 -20283.807} C_VEL
LIN {X 0,Y 250.023,Z 372.163,A -85,B 0,C 180,E1 -20284.394,E2 -20284.394} C_VEL
LIN {X 0,Y 252.67,Z 321.558,A -85,B 0,C 180,E1 -20285.826,E2 -20285.826} C_VEL
LIN {X 0,Y 251.957,Z 318.158,A -85,B 0,C 180,E1 -20286.104,E2 -20286.104} C_VEL
LIN {X 0,Y 246.136,Z 305.133,A -85,B 0,C 180,E1 -20287.874,E2 -20287.874} C_VEL
LIN {X 0,Y 238.906,Z 291.079,A -85,B 0,C 180,E1 -20290.217,E2 -20290.217} C_VEL
LIN {X 0,Y 232.494,Z 280.591,A -85,B 0,C 180,E1 -20292.424,E2 -20292.424} C_VEL
LIN {X 0,Y 229.046,Z 275.285,A -85,B 0,C 180,E1 -20293.69,E2 -20293.69} C_VEL
LIN {X 0,Y 226.011,Z 270.667,A -85,B 0,C 180,E1 -20294.876,E2 -20294.876} C_VEL
LIN {X 0,Y 222.85,Z 265.949,A -85,B 0,C 180,E1 -20296.221,E2 -20296.221} C_VEL
LIN {X 0,Y 222.267,Z 264.258,A -85,B 0,C 180,E1 -20297.208,E2 -20297.208} C_VEL
LIN {X 0,Y 220.817,Z 259.512,A -85,B 0,C 180,E1 -20300.973,E2 -20300.973} C_VEL
LIN {X 0,Y 220.809,Z 259.473,A -85,B 0,C 180,E1 -20305.038,E2 -20305.038} C_VEL
LIN {X 0,Y 220.849,Z 259.472,A -85,B 0,C 180,E1 -20309.384,E2 -20309.384} C_VEL
LIN {X 0,Y 220.868,Z 259.473,A -85,B 0,C 180,E1 -20313.538,E2 -20313.538} C_VEL
LIN {X 0,Y 220.866,Z 259.472,A -85,B 0,C 180,E1 -20317.544,E2 -20317.544} C_VEL
LIN {X 0,Y 220.932,Z 259.465,A -85,B 0,C 180,E1 -20322.617,E2 -20322.617} C_VEL
LIN {X 0,Y 221.007,Z 259.456,A -85,B 0,C 180,E1 -20327.13,E2 -20327.13} C_VEL
LIN {X 0,Y 221.205,Z 259.427,A -85,B 0,C 180,E1 -20330.852,E2 -20330.852} C_VEL
LIN {X 0,Y 221.253,Z 259.416,A -85,B 0,C 180,E1 -20332.692,E2 -20332.692} C_VEL
LIN {X 0,Y 221.476,Z 259.383,A -85,B 0,C 180,E1 -20338.173,E2 -20338.173} C_VEL
LIN {X 0,Y 221.507,Z 259.385,A -85,B 0,C 180,E1 -20341.81,E2 -20341.81} C_VEL
LIN {X 0,Y 221.239,Z 259.413,A -85,B 0,C 180,E1 -20347.292,E2 -20347.292} C_VEL
LIN {X 0,Y 221.062,Z 259.438,A -85,B 0,C 180,E1 -20350.988,E2 -20350.988} C_VEL
LIN {X 0,Y 220.998,Z 259.454,A -85,B 0,C 180,E1 -20356.622,E2 -20356.622} C_VEL
LIN {X 0,Y 220.879,Z 259.473,A -85,B 0,C 180,E1 -20360.478,E2 -20360.478} C_VEL
LIN {X 0,Y 220.899,Z 259.656,A -85,B 0,C 180,E1 -20363.605,E2 -20363.605} C_VEL
LIN {X 0,Y 221.688,Z 261.95,A -85,B 0,C 180,E1 -20365.329,E2 -20365.329} C_VEL
LIN {X 0,Y 224.291,Z 266.063,A -85,B 0,C 180,E1 -20366.552,E2 -20366.552} C_VEL
LIN {X 0,Y 226.232,Z 268.585,A -85,B 0,C 180,E1 -20367.322,E2 -20367.322} C_VEL
LIN {X 0,Y 229.852,Z 273.865,A -85,B 0,C 180,E1 -20368.715,E2 -20368.715} C_VEL
LIN {X 0,Y 235.996,Z 283.249,A -85,B 0,C 180,E1 -20370.901,E2 -20370.901} C_VEL
LIN {X 0,Y 242.619,Z 294.666,A -85,B 0,C 180,E1 -20373.1,E2 -20373.1} C_VEL
LIN {X 0,Y 248.595,Z 306.34,A -85,B 0,C 180,E1 -20374.954,E2 -20374.954} C_VEL
LIN {X 0,Y 252.98,Z 316.256,A -85,B 0,C 180,E1 -20376.267,E2 -20376.267} C_VEL
LIN {X 0,Y 250.007,Z 369.991,A -85,B 0,C 180,E1 -20377.8,E2 -20377.8} C_VEL
LIN {X 0,Y 248.347,Z 383.803,A -85,B 0,C 180,E1 -20378.493,E2 -20378.493} C_VEL
LIN {X 0,Y 246.397,Z 395.728,A -85,B 0,C 180,E1 -20379.408,E2 -20379.408} C_VEL
LIN {X 0,Y 243.934,Z 406.883,A -85,B 0,C 180,E1 -20380.545,E2 -20380.545} C_VEL
LIN {X 0,Y 240.667,Z 419.057,A -85,B 0,C 180,E1 -20382.182,E2 -20382.182} C_VEL
LIN {X 0,Y 237.291,Z 429.882,A -85,B 0,C 180,E1 -20384.091,E2 -20384.091} C_VEL
LIN {X 0,Y 233.829,Z 439.503,A -85,B 0,C 180,E1 -20386.267,E2 -20386.267} C_VEL
LIN {X 0,Y 230.719,Z 447.352,A -85,B 0,C 180,E1 -20388.506,E2 -20388.506} C_VEL
LIN {X 0,Y 227.811,Z 454.193,A -85,B 0,C 180,E1 -20390.961,E2 -20390.961} C_VEL
LIN {X 0,Y 225.102,Z 460.014,A -85,B 0,C 180,E1 -20393.615,E2 -20393.615} C_VEL
LIN {X 0,Y 222.789,Z 464.8,A -85,B 0,C 180,E1 -20396.492,E2 -20396.492} C_VEL
LIN {X 0,Y 220.998,Z 468.352,A -85,B 0,C 180,E1 -20399.414,E2 -20399.414} C_VEL
LIN {X 0,Y 220.063,Z 470.082,A -85,B 0,C 180,E1 -20401.376,E2 -20401.376} C_VEL
LIN {X 0,Y 219.235,Z 471.577,A -85,B 0,C 180,E1 -20403.819,E2 -20403.819} C_VEL
LIN {X 0,Y 218.441,Z 472.485,A -85,B 0,C 180,E1 -20407.289,E2 -20407.289} C_VEL
LIN {X 0,Y 218.274,Z 472.407,A -85,B 0,C 180,E1 -20409.256,E2 -20409.256} C_VEL
LIN {X 0,Y 218.101,Z 471.865,A -85,B 0,C 180,E1 -20411.201,E2 -20411.201} C_VEL
LIN {X 0,Y 218.075,Z 470.883,A -85,B 0,C 180,E1 -20413.139,E2 -20413.139} C_VEL
LIN {X 0,Y 218.214,Z 469.482,A -85,B 0,C 180,E1 -20415.068,E2 -20415.068} C_VEL
LIN {X 0,Y 218.595,Z 466.511,A -85,B 0,C 180,E1 -20417.937,E2 -20417.937} C_VEL
LIN {X 0,Y 219.116,Z 462.472,A -85,B 0,C 180,E1 -20420.771,E2 -20420.771} C_VEL
LIN {X 0,Y 220.152,Z 456.221,A -85,B 0,C 180,E1 -20424.044,E2 -20424.044} C_VEL
LIN {X 0,Y 221.309,Z 449.396,A -85,B 0,C 180,E1 -20426.814,E2 -20426.814} C_VEL
LIN {X 0,Y 222.861,Z 440.914,A -85,B 0,C 180,E1 -20429.548,E2 -20429.548} C_VEL
LIN {X 0,Y 224.507,Z 432.139,A -85,B 0,C 180,E1 -20431.793,E2 -20431.793} C_VEL
LIN {X 0,Y 226.544,Z 421.285,A -85,B 0,C 180,E1 -20434.002,E2 -20434.002} C_VEL
LIN {X 0,Y 228.279,Z 410.501,A -85,B 0,C 180,E1 -20435.742,E2 -20435.742} C_VEL
LIN {X 0,Y 229.933,Z 398.405,A -85,B 0,C 180,E1 -20437.243,E2 -20437.243} C_VEL
LIN {X 0,Y 231.272,Z 385.826,A -85,B 0,C 180,E1 -20438.409,E2 -20438.409} C_VEL
LIN {X 0,Y 232.321,Z 373.618,A -85,B 0,C 180,E1 -20439.193,E2 -20439.193} C_VEL
LIN {X 0,Y 233.025,Z 358.483,A -85,B 0,C 180,E1 -20439.767,E2 -20439.767} C_VEL
LIN {X 0,Y 235.007,Z 302.53,A -85,B 0,C 180,E1 -20441.43,E2 -20441.43} C_VEL
LIN {X 0,Y 233.505,Z 293.685,A -85,B 0,C 180,E1 -20441.888,E2 -20441.888} C_VEL
LIN {X 0,Y 228.638,Z 279.142,A -85,B 0,C 180,E1 -20442.934,E2 -20442.934} C_VEL
LIN {X 0,Y 221.566,Z 261.799,A -85,B 0,C 180,E1 -20444.446,E2 -20444.446} C_VEL
LIN {X 0,Y 221.306,Z 260.796,A -85,B 0,C 180,E1 -20444.717,E2 -20444.717} C_VEL
LIN {X 0,Y 221.03,Z 259.513,A -85,B 0,C 180,E1 -20445.443,E2 -20445.443} C_VEL
LIN {X 0,Y 220.904,Z 259.439,A -85,B 0,C 180,E1 -20448.55,E2 -20448.55} C_VEL
LIN {X 0,Y 220.901,Z 259.47,A -85,B 0,C 180,E1 -20452.713,E2 -20452.713} C_VEL
LIN {X 0,Y 220.856,Z 259.423,A -85,B 0,C 180,E1 -20457.023,E2 -20457.023} C_VEL
LIN {X 0,Y 220.859,Z 259.471,A -85,B 0,C 180,E1 -20460.797,E2 -20460.797} C_VEL
LIN {X 0,Y 220.84,Z 259.459,A -85,B 0,C 180,E1 -20464.947,E2 -20464.947} C_VEL
LIN {X 0,Y 220.854,Z 259.471,A -85,B 0,C 180,E1 -20469.526,E2 -20469.526} C_VEL
LIN {X 0,Y 220.867,Z 259.447,A -85,B 0,C 180,E1 -20472.972,E2 -20472.972} C_VEL
LIN {X 0,Y 220.864,Z 259.472,A -85,B 0,C 180,E1 -20477.042,E2 -20477.042} C_VEL
LIN {X 0,Y 220.834,Z 259.443,A -85,B 0,C 180,E1 -20480.482,E2 -20480.482} C_VEL
LIN {X 0,Y 220.792,Z 259.479,A -85,B 0,C 180,E1 -20485.055,E2 -20485.055} C_VEL
LIN {X 0,Y 220.847,Z 259.458,A -85,B 0,C 180,E1 -20489.403,E2 -20489.403} C_VEL
LIN {X 0,Y 220.877,Z 259.431,A -85,B 0,C 180,E1 -20493.558,E2 -20493.558} C_VEL
LIN {X 0,Y 220.92,Z 259.465,A -85,B 0,C 180,E1 -20497.568,E2 -20497.568} C_VEL
LIN {X 0,Y 220.98,Z 259.424,A -85,B 0,C 180,E1 -20502.573,E2 -20502.573} C_VEL
LIN {X 0,Y 221.003,Z 259.424,A -85,B 0,C 180,E1 -20507.147,E2 -20507.147} C_VEL
LIN {X 0,Y 221.25,Z 259.423,A -85,B 0,C 180,E1 -20510.87,E2 -20510.87} C_VEL
LIN {X 0,Y 221.305,Z 259.415,A -85,B 0,C 180,E1 -20512.711,E2 -20512.711} C_VEL
LIN {X 0,Y 221.508,Z 259.341,A -85,B 0,C 180,E1 -20518.19,E2 -20518.19} C_VEL
LIN {X 0,Y 221.509,Z 259.381,A -85,B 0,C 180,E1 -20521.826,E2 -20521.826} C_VEL
LIN {X 0,Y 221.242,Z 259.407,A -85,B 0,C 180,E1 -20527.308,E2 -20527.308} C_VEL
LIN {X 0,Y 221.069,Z 259.405,A -85,B 0,C 180,E1 -20531.004,E2 -20531.004} C_VEL
LIN {X 0,Y 221,Z 259.455,A -85,B 0,C 180,E1 -20534.746,E2 -20534.746} C_VEL
LIN {X 0,Y 220.927,Z 259.45,A -85,B 0,C 180,E1 -20538.557,E2 -20538.557} C_VEL
LIN {X 0,Y 220.893,Z 259.447,A -85,B 0,C 180,E1 -20542.682,E2 -20542.682} C_VEL
LIN {X 0,Y 220.889,Z 259.467,A -85,B 0,C 180,E1 -20547.019,E2 -20547.019} C_VEL
LIN {X 0,Y 220.829,Z 259.456,A -85,B 0,C 180,E1 -20550.765,E2 -20550.765} C_VEL
LIN {X 0,Y 220.805,Z 259.479,A -85,B 0,C 180,E1 -20554.962,E2 -20554.962} C_VEL
LIN {X 0,Y 220.81,Z 259.463,A -85,B 0,C 180,E1 -20556.858,E2 -20556.858} C_VEL
LIN {X 0,Y 220.204,Z 259.545,A -85,B 0,C 180,E1 -20558.379,E2 -20558.379} C_VEL
LIN {X 0,Y 218.621,Z 259.754,A -85,B 0,C 180,E1 -20559.872,E2 -20559.872} C_VEL
LIN {X 0,Y 214.819,Z 260.197,A -85,B 0,C 180,E1 -20562.883,E2 -20562.883} C_VEL
LIN {X 0,Y 213.745,Z 260.309,A -85,B 0,C 180,E1 -20564.458,E2 -20564.458} C_VEL
LIN {X 0,Y 213.66,Z 260.317,A -85,B 0,C 180,E1 -20564.993,E2 -20564.993} C_VEL
LIN {X 0,Y 213.717,Z 260.363,A -85,B 0,C 180,E1 -20569.153,E2 -20569.153} C_VEL
LIN {X 0,Y 213.798,Z 260.411,A -85,B 0,C 180,E1 -20573.723,E2 -20573.723} C_VEL
LIN {X 0,Y 215.034,Z 265.821,A -85,B 0,C 180,E1 -20576.402,E2 -20576.402} C_VEL
LIN {X 0,Y 215.285,Z 266.946,A -85,B 0,C 180,E1 -20576.743,E2 -20576.743} C_VEL
LIN {X 0,Y 222.611,Z 285.579,A -85,B 0,C 180,E1 -20578.407,E2 -20578.407} C_VEL
LIN {X 0,Y 225.559,Z 294.695,A -85,B 0,C 180,E1 -20579.085,E2 -20579.085} C_VEL
LIN {X 0,Y 228.137,Z 316.109,A -85,B 0,C 180,E1 -20580.123,E2 -20580.123} C_VEL
LIN {X 0,Y 226.032,Z 375.228,A -85,B 0,C 180,E1 -20581.999,E2 -20581.999} C_VEL
LIN {X 0,Y 225.005,Z 387.586,A -85,B 0,C 180,E1 -20582.694,E2 -20582.694} C_VEL
LIN {X 0,Y 223.591,Z 400.388,A -85,B 0,C 180,E1 -20583.768,E2 -20583.768} C_VEL
LIN {X 0,Y 221.829,Z 412.547,A -85,B 0,C 180,E1 -20585.18,E2 -20585.18} C_VEL
LIN {X 0,Y 219.827,Z 424.126,A -85,B 0,C 180,E1 -20586.944,E2 -20586.944} C_VEL
LIN {X 0,Y 218.051,Z 434.587,A -85,B 0,C 180,E1 -20588.988,E2 -20588.988} C_VEL
LIN {X 0,Y 216.531,Z 443.114,A -85,B 0,C 180,E1 -20591.061,E2 -20591.061} C_VEL
LIN {X 0,Y 214.936,Z 450.934,A -85,B 0,C 180,E1 -20593.376,E2 -20593.376} C_VEL
LIN {X 0,Y 213.399,Z 458.562,A -85,B 0,C 180,E1 -20596.187,E2 -20596.187} C_VEL
LIN {X 0,Y 212.309,Z 465.605,A -85,B 0,C 180,E1 -20599.511,E2 -20599.511} C_VEL
LIN {X 0,Y 211.706,Z 470.234,A -85,B 0,C 180,E1 -20602.37,E2 -20602.37} C_VEL
LIN {X 0,Y 211.507,Z 472.668,A -85,B 0,C 180,E1 -20604.28,E2 -20604.28} C_VEL
LIN {X 0,Y 211.378,Z 474.65,A -85,B 0,C 180,E1 -20606.188,E2 -20606.188} C_VEL
LIN {X 0,Y 211.388,Z 476.214,A -85,B 0,C 180,E1 -20608.095,E2 -20608.095} C_VEL
LIN {X 0,Y 211.466,Z 477.342,A -85,B 0,C 180,E1 -20610.001,E2 -20610.001} C_VEL
LIN {X 0,Y 211.39,Z 478.038,A -85,B 0,C 180,E1 -20611.906,E2 -20611.906} C_VEL
LIN {X 0,Y 211.587,Z 478.286,A -85,B 0,C 180,E1 -20615.719,E2 -20615.719} C_VEL
LIN {X 0,Y 211.847,Z 477.831,A -85,B 0,C 180,E1 -20617.626,E2 -20617.626} C_VEL
LIN {X 0,Y 212.919,Z 475.692,A -85,B 0,C 180,E1 -20621.423,E2 -20621.423} C_VEL
LIN {X 0,Y 214.289,Z 473.036,A -85,B 0,C 180,E1 -20624.24,E2 -20624.24} C_VEL
LIN {X 0,Y 216.049,Z 469.395,A -85,B 0,C 180,E1 -20627.024,E2 -20627.024} C_VEL
LIN {X 0,Y 218.48,Z 464.667,A -85,B 0,C 180,E1 -20629.741,E2 -20629.741} C_VEL
LIN {X 0,Y 221.266,Z 458.721,A -85,B 0,C 180,E1 -20632.406,E2 -20632.406} C_VEL
LIN {X 0,Y 224.393,Z 451.353,A -85,B 0,C 180,E1 -20635.013,E2 -20635.013} C_VEL
LIN {X 0,Y 227.489,Z 443.852,A -85,B 0,C 180,E1 -20637.109,E2 -20637.109} C_VEL
LIN {X 0,Y 230.986,Z 434.785,A -85,B 0,C 180,E1 -20639.132,E2 -20639.132} C_VEL
LIN {X 0,Y 234.357,Z 424.756,A -85,B 0,C 180,E1 -20640.901,E2 -20640.901} C_VEL
LIN {X 0,Y 237.137,Z 415.227,A -85,B 0,C 180,E1 -20642.24,E2 -20642.24} C_VEL
LIN {X 0,Y 240.047,Z 403.216,A -85,B 0,C 180,E1 -20643.547,E2 -20643.547} C_VEL
LIN {X 0,Y 242.463,Z 390.695,A -85,B 0,C 180,E1 -20644.544,E2 -20644.544} C_VEL
LIN {X 0,Y 244.218,Z 377.345,A -85,B 0,C 180,E1 -20645.268,E2 -20645.268} C_VEL
LIN {X 0,Y 245.43,Z 359.091,A -85,B 0,C 180,E1 -20645.858,E2 -20645.858} C_VEL
LIN {X 0,Y 247.376,Z 322.932,A -85,B 0,C 180,E1 -20646.882,E2 -20646.882} C_VEL
LIN {X 0,Y 246.416,Z 319.969,A -85,B 0,C 180,E1 -20647.21,E2 -20647.21} C_VEL
LIN {X 0,Y 241.21,Z 308.359,A -85,B 0,C 180,E1 -20648.89,E2 -20648.89} C_VEL
LIN {X 0,Y 234.841,Z 295.74,A -85,B 0,C 180,E1 -20651.077,E2 -20651.077} C_VEL
LIN {X 0,Y 228.667,Z 285.472,A -85,B 0,C 180,E1 -20653.31,E2 -20653.31} C_VEL
LIN {X 0,Y 225.59,Z 280.613,A -85,B 0,C 180,E1 -20654.496,E2 -20654.496} C_VEL
LIN {X 0,Y 222.553,Z 275.957,A -85,B 0,C 180,E1 -20655.738,E2 -20655.738} C_VEL
LIN {X 0,Y 218.809,Z 270.567,A -85,B 0,C 180,E1 -20657.35,E2 -20657.35} C_VEL
LIN {X 0,Y 215.539,Z 265.873,A -85,B 0,C 180,E1 -20658.912,E2 -20658.912} C_VEL
LIN {X 0,Y 214.97,Z 264.434,A -85,B 0,C 180,E1 -20659.774,E2 -20659.774} C_VEL
LIN {X 0,Y 213.791,Z 260.398,A -85,B 0,C 180,E1 -20663.325,E2 -20663.325} C_VEL
LIN {X 0,Y 213.774,Z 260.347,A -85,B 0,C 180,E1 -20668.255,E2 -20668.255} C_VEL
LIN {X 0,Y 213.797,Z 260.345,A -85,B 0,C 180,E1 -20672.591,E2 -20672.591} C_VEL
LIN {X 0,Y 213.791,Z 260.347,A -85,B 0,C 180,E1 -20676.993,E2 -20676.993} C_VEL
LIN {X 0,Y 213.896,Z 260.338,A -85,B 0,C 180,E1 -20682.792,E2 -20682.792} C_VEL
LIN {X 0,Y 213.946,Z 260.335,A -85,B 0,C 180,E1 -20686.698,E2 -20686.698} C_VEL
LIN {X 0,Y 214.144,Z 260.302,A -85,B 0,C 180,E1 -20690.547,E2 -20690.547} C_VEL
LIN {X 0,Y 214.087,Z 260.303,A -85,B 0,C 180,E1 -20694.34,E2 -20694.34} C_VEL
LIN {X 0,Y 214.413,Z 260.262,A -85,B 0,C 180,E1 -20698.113,E2 -20698.113} C_VEL
LIN {X 0,Y 214.542,Z 260.254,A -85,B 0,C 180,E1 -20699.992,E2 -20699.992} C_VEL
LIN {X 0,Y 214.44,Z 260.264,A -85,B 0,C 180,E1 -20701.87,E2 -20701.87} C_VEL
LIN {X 0,Y 214.18,Z 260.292,A -85,B 0,C 180,E1 -20707.533,E2 -20707.533} C_VEL
LIN {X 0,Y 213.993,Z 260.317,A -85,B 0,C 180,E1 -20711.356,E2 -20711.356} C_VEL
LIN {X 0,Y 213.913,Z 260.329,A -85,B 0,C 180,E1 -20715.229,E2 -20715.229} C_VEL
LIN {X 0,Y 213.826,Z 260.342,A -85,B 0,C 180,E1 -20719.179,E2 -20719.179} C_VEL
LIN {X 0,Y 213.82,Z 260.487,A -85,B 0,C 180,E1 -20721.186,E2 -20721.186} C_VEL
LIN {X 0,Y 214.434,Z 262.468,A -85,B 0,C 180,E1 -20722.667,E2 -20722.667} C_VEL
LIN {X 0,Y 218.211,Z 267.448,A -85,B 0,C 180,E1 -20724.488,E2 -20724.488} C_VEL
LIN {X 0,Y 222.193,Z 272.897,A -85,B 0,C 180,E1 -20726.211,E2 -20726.211} C_VEL
LIN {X 0,Y 226.536,Z 279.44,A -85,B 0,C 180,E1 -20727.974,E2 -20727.974} C_VEL
LIN {X 0,Y 232.251,Z 288.353,A -85,B 0,C 180,E1 -20730.099,E2 -20730.099} C_VEL
LIN {X 0,Y 238.529,Z 299.363,A -85,B 0,C 180,E1 -20732.286,E2 -20732.286} C_VEL
LIN {X 0,Y 244.673,Z 311.711,A -85,B 0,C 180,E1 -20734.302,E2 -20734.302} C_VEL
LIN {X 0,Y 247.581,Z 318.42,A -85,B 0,C 180,E1 -20735.217,E2 -20735.217} C_VEL
LIN {X 0,Y 244.728,Z 369.503,A -85,B 0,C 180,E1 -20736.704,E2 -20736.704} C_VEL
LIN {X 0,Y 243.152,Z 382.49,A -85,B 0,C 180,E1 -20737.342,E2 -20737.342} C_VEL
LIN {X 0,Y 241.114,Z 394.797,A -85,B 0,C 180,E1 -20738.263,E2 -20738.263} C_VEL
LIN {X 0,Y 238.625,Z 405.863,A -85,B 0,C 180,E1 -20739.365,E2 -20739.365} C_VEL
LIN {X 0,Y 235.367,Z 417.775,A -85,B 0,C 180,E1 -20740.951,E2 -20740.951} C_VEL
LIN {X 0,Y 232.062,Z 428.161,A -85,B 0,C 180,E1 -20742.742,E2 -20742.742} C_VEL
LIN {X 0,Y 228.38,Z 438.159,A -85,B 0,C 180,E1 -20744.944,E2 -20744.944} C_VEL
LIN {X 0,Y 225.026,Z 446.243,A -85,B 0,C 180,E1 -20747.211,E2 -20747.211} C_VEL
LIN {X 0,Y 221.654,Z 453.812,A -85,B 0,C 180,E1 -20749.915,E2 -20749.915} C_VEL
LIN {X 0,Y 218.955,Z 459.316,A -85,B 0,C 180,E1 -20752.42,E2 -20752.42} C_VEL
LIN {X 0,Y 216.436,Z 464.315,A -85,B 0,C 180,E1 -20755.371,E2 -20755.371} C_VEL
LIN {X 0,Y 214.388,Z 468.122,A -85,B 0,C 180,E1 -20758.445,E2 -20758.445} C_VEL
LIN {X 0,Y 213.36,Z 469.862,A -85,B 0,C 180,E1 -20760.389,E2 -20760.389} C_VEL
LIN {X 0,Y 212.257,Z 471.686,A -85,B 0,C 180,E1 -20763.355,E2 -20763.355} C_VEL
LIN {X 0,Y 211.467,Z 472.554,A -85,B 0,C 180,E1 -20766.495,E2 -20766.495} C_VEL
LIN {X 0,Y 211.22,Z 472.534,A -85,B 0,C 180,E1 -20768.664,E2 -20768.664} C_VEL
LIN {X 0,Y 211.042,Z 472.123,A -85,B 0,C 180,E1 -20770.548,E2 -20770.548} C_VEL
LIN {X 0,Y 210.985,Z 471.227,A -85,B 0,C 180,E1 -20772.554,E2 -20772.554} C_VEL
LIN {X 0,Y 211.109,Z 469.668,A -85,B 0,C 180,E1 -20774.849,E2 -20774.849} C_VEL
LIN {X 0,Y 211.444,Z 467.066,A -85,B 0,C 180,E1 -20777.522,E2 -20777.522} C_VEL
LIN {X 0,Y 211.953,Z 463.175,A -85,B 0,C 180,E1 -20780.456,E2 -20780.456} C_VEL
LIN {X 0,Y 212.815,Z 457.87,A -85,B 0,C 180,E1 -20783.489,E2 -20783.489} C_VEL
LIN {X 0,Y 213.927,Z 451.749,A -85,B 0,C 180,E1 -20786.232,E2 -20786.232} C_VEL
LIN {X 0,Y 215.381,Z 443.776,A -85,B 0,C 180,E1 -20789.065,E2 -20789.065} C_VEL
LIN {X 0,Y 216.956,Z 435.617,A -85,B 0,C 180,E1 -20791.392,E2 -20791.392} C_VEL
LIN {X 0,Y 218.883,Z 425.639,A -85,B 0,C 180,E1 -20793.681,E2 -20793.681} C_VEL
LIN {X 0,Y 220.629,Z 415.831,A -85,B 0,C 180,E1 -20795.483,E2 -20795.483} C_VEL
LIN {X 0,Y 222.318,Z 405.216,A -85,B 0,C 180,E1 -20797.036,E2 -20797.036} C_VEL
LIN {X 0,Y 223.939,Z 392.456,A -85,B 0,C 180,E1 -20798.459,E2 -20798.459} C_VEL
LIN {X 0,Y 225.219,Z 379.684,A -85,B 0,C 180,E1 -20799.485,E2 -20799.485} C_VEL
LIN {X 0,Y 226.083,Z 367.445,A -85,B 0,C 180,E1 -20800.126,E2 -20800.126} C_VEL
LIN {X 0,Y 228.441,Z 302.996,A -85,B 0,C 180,E1 -20802.13,E2 -20802.13} C_VEL
LIN {X 0,Y 227.072,Z 295.275,A -85,B 0,C 180,E1 -20802.554,E2 -20802.554} C_VEL
LIN {X 0,Y 222.285,Z 281.221,A -85,B 0,C 180,E1 -20803.623,E2 -20803.623} C_VEL
LIN {X 0,Y 215.308,Z 264.221,A -85,B 0,C 180,E1 -20805.155,E2 -20805.155} C_VEL
LIN {X 0,Y 214.174,Z 261.386,A -85,B 0,C 180,E1 -20805.523,E2 -20805.523} C_VEL
LIN {X 0,Y 213.971,Z 260.439,A -85,B 0,C 180,E1 -20805.966,E2 -20805.966} C_VEL
LIN {X 0,Y 213.851,Z 260.315,A -85,B 0,C 180,E1 -20809.186,E2 -20809.186} C_VEL
LIN {X 0,Y 213.825,Z 260.348,A -85,B 0,C 180,E1 -20813.229,E2 -20813.229} C_VEL
LIN {X 0,Y 213.793,Z 260.303,A -85,B 0,C 180,E1 -20817.454,E2 -20817.454} C_VEL
LIN {X 0,Y 213.773,Z 260.361,A -85,B 0,C 180,E1 -20821.736,E2 -20821.736} C_VEL
LIN {X 0,Y 213.762,Z 260.344,A -85,B 0,C 180,E1 -20826.284,E2 -20826.284} C_VEL
LIN {X 0,Y 213.804,Z 260.332,A -85,B 0,C 180,E1 -20831.103,E2 -20831.103} C_VEL
LIN {X 0,Y 213.807,Z 260.331,A -85,B 0,C 180,E1 -20833.699,E2 -20833.699} C_VEL
LIN {X 0,Y 213.812,Z 260.352,A -85,B 0,C 180,E1 -20836.363,E2 -20836.363} C_VEL
LIN {X 0,Y 213.797,Z 260.335,A -85,B 0,C 180,E1 -20839.117,E2 -20839.117} C_VEL
LIN {X 0,Y 213.73,Z 260.345,A -85,B 0,C 180,E1 -20843.721,E2 -20843.721} C_VEL
LIN {X 0,Y 213.775,Z 260.345,A -85,B 0,C 180,E1 -20848.732,E2 -20848.732} C_VEL
LIN {X 0,Y 213.807,Z 260.305,A -85,B 0,C 180,E1 -20852.612,E2 -20852.612} C_VEL
LIN {X 0,Y 213.85,Z 260.342,A -85,B 0,C 180,E1 -20856.952,E2 -20856.952} C_VEL
LIN {X 0,Y 213.957,Z 260.295,A -85,B 0,C 180,E1 -20862.814,E2 -20862.814} C_VEL
LIN {X 0,Y 214.033,Z 260.31,A -85,B 0,C 180,E1 -20868.647,E2 -20868.647} C_VEL
LIN {X 0,Y 214.241,Z 260.295,A -85,B 0,C 180,E1 -20872.469,E2 -20872.469} C_VEL
LIN {X 0,Y 214.441,Z 260.22,A -85,B 0,C 180,E1 -20878.13,E2 -20878.13} C_VEL
LIN {X 0,Y 214.544,Z 260.225,A -85,B 0,C 180,E1 -20880.008,E2 -20880.008} C_VEL
LIN {X 0,Y 214.442,Z 260.261,A -85,B 0,C 180,E1 -20881.886,E2 -20881.886} C_VEL
LIN {X 0,Y 214.184,Z 260.282,A -85,B 0,C 180,E1 -20887.55,E2 -20887.55} C_VEL
LIN {X 0,Y 214.001,Z 260.287,A -85,B 0,C 180,E1 -20891.372,E2 -20891.372} C_VEL
LIN {X 0,Y 213.938,Z 260.334,A -85,B 0,C 180,E1 -20895.245,E2 -20895.245} C_VEL
LIN {X 0,Y 213.842,Z 260.324,A -85,B 0,C 180,E1 -20899.195,E2 -20899.195} C_VEL
LIN {X 0,Y 213.819,Z 260.334,A -85,B 0,C 180,E1 -20903.238,E2 -20903.238} C_VEL
LIN {X 0,Y 213.821,Z 260.346,A -85,B 0,C 180,E1 -20907.447,E2 -20907.447} C_VEL
LIN {X 0,Y 213.77,Z 260.346,A -85,B 0,C 180,E1 -20911.745,E2 -20911.745} C_VEL
LIN {X 0,Y 213.754,Z 260.345,A -85,B 0,C 180,E1 -20916.295,E2 -20916.295} C_VEL
LIN {X 0,Y 213.724,Z 260.358,A -85,B 0,C 180,E1 -20921.131,E2 -20921.131} C_VEL
LIN {X 0,Y 213.66,Z 260.317,A -85,B 0,C 180,E1 -20924.993,E2 -20924.993} C_VEL
LIN {X 0,Y 212.988,Z 260.407,A -85,B 0,C 180,E1 -20926.039,E2 -20926.039} C_VEL
LIN {X 0,Y 210.164,Z 260.783,A -85,B 0,C 180,E1 -20927.685,E2 -20927.685} C_VEL
LIN {X 0,Y 207.315,Z 261.162,A -85,B 0,C 180,E1 -20929.373,E2 -20929.373} C_VEL
LIN {X 0,Y 206.648,Z 261.234,A -85,B 0,C 180,E1 -20930.468,E2 -20930.468} C_VEL
LIN {X 0,Y 206.792,Z 261.368,A -85,B 0,C 180,E1 -20933.183,E2 -20933.183} C_VEL
LIN {X 0,Y 207.974,Z 266.517,A -85,B 0,C 180,E1 -20935.67,E2 -20935.67} C_VEL
LIN {X 0,Y 214.763,Z 283.396,A -85,B 0,C 180,E1 -20937.324,E2 -20937.324} C_VEL
LIN {X 0,Y 219.29,Z 296.642,A -85,B 0,C 180,E1 -20938.394,E2 -20938.394} C_VEL
LIN {X 0,Y 221.658,Z 316.528,A -85,B 0,C 180,E1 -20939.399,E2 -20939.399} C_VEL
LIN {X 0,Y 219.468,Z 374.76,A -85,B 0,C 180,E1 -20941.293,E2 -20941.293} C_VEL
LIN {X 0,Y 218.433,Z 387.097,A -85,B 0,C 180,E1 -20941.996,E2 -20941.996} C_VEL
LIN {X 0,Y 217.057,Z 399.435,A -85,B 0,C 180,E1 -20943.045,E2 -20943.045} C_VEL
LIN {X 0,Y 215.4,Z 411.032,A -85,B 0,C 180,E1 -20944.386,E2 -20944.386} C_VEL
LIN {X 0,Y 213.242,Z 422.879,A -85,B 0,C 180,E1 -20946.189,E2 -20946.189} C_VEL
LIN {X 0,Y 211.383,Z 433.544,A -85,B 0,C 180,E1 -20948.293,E2 -20948.293} C_VEL
LIN {X 0,Y 209.966,Z 440.753,A -85,B 0,C 180,E1 -20950.03,E2 -20950.03} C_VEL
LIN {X 0,Y 208.08,Z 450.211,A -85,B 0,C 180,E1 -20952.811,E2 -20952.811} C_VEL
LIN {X 0,Y 206.482,Z 457.97,A -85,B 0,C 180,E1 -20955.714,E2 -20955.714} C_VEL
LIN {X 0,Y 205.283,Z 465.106,A -85,B 0,C 180,E1 -20959.147,E2 -20959.147} C_VEL
LIN {X 0,Y 204.66,Z 469.826,A -85,B 0,C 180,E1 -20962.106,E2 -20962.106} C_VEL
LIN {X 0,Y 204.346,Z 473.405,A -85,B 0,C 180,E1 -20965.068,E2 -20965.068} C_VEL
LIN {X 0,Y 204.296,Z 475.956,A -85,B 0,C 180,E1 -20968.029,E2 -20968.029} C_VEL
LIN {X 0,Y 204.369,Z 477.145,A -85,B 0,C 180,E1 -20970.001,E2 -20970.001} C_VEL
LIN {X 0,Y 204.298,Z 477.886,A -85,B 0,C 180,E1 -20971.972,E2 -20971.972} C_VEL
LIN {X 0,Y 204.518,Z 478.204,A -85,B 0,C 180,E1 -20975.918,E2 -20975.918} C_VEL
LIN {X 0,Y 204.787,Z 477.796,A -85,B 0,C 180,E1 -20977.891,E2 -20977.891} C_VEL
LIN {X 0,Y 205.267,Z 476.979,A -85,B 0,C 180,E1 -20979.858,E2 -20979.858} C_VEL
LIN {X 0,Y 206.872,Z 474.132,A -85,B 0,C 180,E1 -20983.758,E2 -20983.758} C_VEL
LIN {X 0,Y 208.591,Z 470.898,A -85,B 0,C 180,E1 -20986.642,E2 -20986.642} C_VEL
LIN {X 0,Y 210.915,Z 466.624,A -85,B 0,C 180,E1 -20989.465,E2 -20989.465} C_VEL
LIN {X 0,Y 214.26,Z 460.193,A -85,B 0,C 180,E1 -20992.67,E2 -20992.67} C_VEL
LIN {X 0,Y 217.394,Z 453.185,A -85,B 0,C 180,E1 -20995.363,E2 -20995.363} C_VEL
LIN {X 0,Y 221.234,Z 444.457,A -85,B 0,C 180,E1 -20997.942,E2 -20997.942} C_VEL
LIN {X 0,Y 225.257,Z 434.558,A -85,B 0,C 180,E1 -21000.206,E2 -21000.206} C_VEL
LIN {X 0,Y 228.744,Z 424.494,A -85,B 0,C 180,E1 -21002.006,E2 -21002.006} C_VEL
LIN {X 0,Y 231.643,Z 414.927,A -85,B 0,C 180,E1 -21003.361,E2 -21003.361} C_VEL
LIN {X 0,Y 234.679,Z 402.859,A -85,B 0,C 180,E1 -21004.681,E2 -21004.681} C_VEL
LIN {X 0,Y 237.184,Z 390.255,A -85,B 0,C 180,E1 -21005.688,E2 -21005.688} C_VEL
LIN {X 0,Y 238.967,Z 376.985,A -85,B 0,C 180,E1 -21006.406,E2 -21006.406} C_VEL
LIN {X 0,Y 240.293,Z 357.498,A -85,B 0,C 180,E1 -21007.034,E2 -21007.034} C_VEL
LIN {X 0,Y 242.138,Z 324.642,A -85,B 0,C 180,E1 -21007.977,E2 -21007.977} C_VEL
LIN {X 0,Y 236.828,Z 312.438,A -85,B 0,C 180,E1 -21009.802,E2 -21009.802} C_VEL
LIN {X 0,Y 230.956,Z 300.61,A -85,B 0,C 180,E1 -21011.92,E2 -21011.92} C_VEL
LIN {X 0,Y 225.094,Z 290.638,A -85,B 0,C 180,E1 -21014.15,E2 -21014.15} C_VEL
LIN {X 0,Y 222.244,Z 286.026,A -85,B 0,C 180,E1 -21015.301,E2 -21015.301} C_VEL
LIN {X 0,Y 219.183,Z 281.268,A -85,B 0,C 180,E1 -21016.612,E2 -21016.612} C_VEL
LIN {X 0,Y 215.653,Z 276.116,A -85,B 0,C 180,E1 -21018.213,E2 -21018.213} C_VEL
LIN {X 0,Y 211.706,Z 270.572,A -85,B 0,C 180,E1 -21020.152,E2 -21020.152} C_VEL
LIN {X 0,Y 208.059,Z 265.445,A -85,B 0,C 180,E1 -21022.182,E2 -21022.182} C_VEL
LIN {X 0,Y 207.458,Z 263.567,A -85,B 0,C 180,E1 -21023.633,E2 -21023.633} C_VEL
LIN {X 0,Y 206.735,Z 261.256,A -85,B 0,C 180,E1 -21026.165,E2 -21026.165} C_VEL
LIN {X 0,Y 206.71,Z 261.232,A -85,B 0,C 180,E1 -21029.328,E2 -21029.328} C_VEL
LIN {X 0,Y 206.698,Z 261.239,A -85,B 0,C 180,E1 -21033.759,E2 -21033.759} C_VEL
LIN {X 0,Y 206.721,Z 261.236,A -85,B 0,C 180,E1 -21038.031,E2 -21038.031} C_VEL
LIN {X 0,Y 206.832,Z 261.222,A -85,B 0,C 180,E1 -21042.185,E2 -21042.185} C_VEL
LIN {X 0,Y 206.886,Z 261.21,A -85,B 0,C 180,E1 -21046.235,E2 -21046.235} C_VEL
LIN {X 0,Y 207.087,Z 261.178,A -85,B 0,C 180,E1 -21050.222,E2 -21050.222} C_VEL
LIN {X 0,Y 207.05,Z 261.179,A -85,B 0,C 180,E1 -21054.147,E2 -21054.147} C_VEL
LIN {X 0,Y 207.352,Z 261.142,A -85,B 0,C 180,E1 -21058.049,E2 -21058.049} C_VEL
LIN {X 0,Y 207.507,Z 261.13,A -85,B 0,C 180,E1 -21059.991,E2 -21059.991} C_VEL
LIN {X 0,Y 207.376,Z 261.143,A -85,B 0,C 180,E1 -21061.933,E2 -21061.933} C_VEL
LIN {X 0,Y 207.125,Z 261.172,A -85,B 0,C 180,E1 -21067.791,E2 -21067.791} C_VEL
LIN {X 0,Y 206.916,Z 261.199,A -85,B 0,C 180,E1 -21071.749,E2 -21071.749} C_VEL
LIN {X 0,Y 206.848,Z 261.21,A -85,B 0,C 180,E1 -21075.762,E2 -21075.762} C_VEL
LIN {X 0,Y 206.836,Z 261.465,A -85,B 0,C 180,E1 -21078.609,E2 -21078.609} C_VEL
LIN {X 0,Y 207.198,Z 262.862,A -85,B 0,C 180,E1 -21079.495,E2 -21079.495} C_VEL
LIN {X 0,Y 208.757,Z 265.307,A -85,B 0,C 180,E1 -21080.433,E2 -21080.433} C_VEL
LIN {X 0,Y 211.896,Z 268.849,A -85,B 0,C 180,E1 -21082.053,E2 -21082.053} C_VEL
LIN {X 0,Y 216.314,Z 274.754,A -85,B 0,C 180,E1 -21084.194,E2 -21084.194} C_VEL
LIN {X 0,Y 220.157,Z 280.316,A -85,B 0,C 180,E1 -21085.914,E2 -21085.914} C_VEL
LIN {X 0,Y 223.343,Z 285.158,A -85,B 0,C 180,E1 -21087.246,E2 -21087.246} C_VEL
LIN {X 0,Y 229.029,Z 294.287,A -85,B 0,C 180,E1 -21089.457,E2 -21089.457} C_VEL
LIN {X 0,Y 234.691,Z 304.432,A -85,B 0,C 180,E1 -21091.515,E2 -21091.515} C_VEL
LIN {X 0,Y 240.548,Z 316.515,A -85,B 0,C 180,E1 -21093.534,E2 -21093.534} C_VEL
LIN {X 0,Y 242.374,Z 320.879,A -85,B 0,C 180,E1 -21094.154,E2 -21094.154} C_VEL
LIN {X 0,Y 239.467,Z 369.417,A -85,B 0,C 180,E1 -21095.569,E2 -21095.569} C_VEL
LIN {X 0,Y 237.799,Z 382.796,A -85,B 0,C 180,E1 -21096.236,E2 -21096.236} C_VEL
LIN {X 0,Y 235.783,Z 394.527,A -85,B 0,C 180,E1 -21097.123,E2 -21097.123} C_VEL
LIN {X 0,Y 232.97,Z 406.556,A -85,B 0,C 180,E1 -21098.34,E2 -21098.34} C_VEL
LIN {X 0,Y 229.874,Z 417.453,A -85,B 0,C 180,E1 -21099.811,E2 -21099.811} C_VEL
LIN {X 0,Y 226.139,Z 428.646,A -85,B 0,C 180,E1 -21101.765,E2 -21101.765} C_VEL
LIN {X 0,Y 222.453,Z 438.217,A -85,B 0,C 180,E1 -21103.923,E2 -21103.923} C_VEL
LIN {X 0,Y 218.799,Z 446.585,A -85,B 0,C 180,E1 -21106.322,E2 -21106.322} C_VEL
LIN {X 0,Y 215.127,Z 454.387,A -85,B 0,C 180,E1 -21109.203,E2 -21109.203} C_VEL
LIN {X 0,Y 211.928,Z 460.505,A -85,B 0,C 180,E1 -21112.157,E2 -21112.157} C_VEL
LIN {X 0,Y 209.341,Z 465.219,A -85,B 0,C 180,E1 -21115.199,E2 -21115.199} C_VEL
LIN {X 0,Y 207.581,Z 468.256,A -85,B 0,C 180,E1 -21117.803,E2 -21117.803} C_VEL
LIN {X 0,Y 205.798,Z 471.074,A -85,B 0,C 180,E1 -21121.438,E2 -21121.438} C_VEL
LIN {X 0,Y 205.085,Z 472.068,A -85,B 0,C 180,E1 -21123.545,E2 -21123.545} C_VEL
LIN {X 0,Y 204.52,Z 472.62,A -85,B 0,C 180,E1 -21125.646,E2 -21125.646} C_VEL
LIN {X 0,Y 204.14,Z 472.634,A -85,B 0,C 180,E1 -21128.332,E2 -21128.332} C_VEL
LIN {X 0,Y 203.894,Z 471.561,A -85,B 0,C 180,E1 -21131.927,E2 -21131.927} C_VEL
LIN {X 0,Y 203.986,Z 469.8,A -85,B 0,C 180,E1 -21134.686,E2 -21134.686} C_VEL
LIN {X 0,Y 204.407,Z 466.515,A -85,B 0,C 180,E1 -21138.094,E2 -21138.094} C_VEL
LIN {X 0,Y 204.978,Z 462.406,A -85,B 0,C 180,E1 -21141.124,E2 -21141.124} C_VEL
LIN {X 0,Y 205.932,Z 457.086,A -85,B 0,C 180,E1 -21144.123,E2 -21144.123} C_VEL
LIN {X 0,Y 207.163,Z 450.399,A -85,B 0,C 180,E1 -21147.082,E2 -21147.082} C_VEL
LIN {X 0,Y 208.766,Z 442.093,A -85,B 0,C 180,E1 -21149.999,E2 -21149.999} C_VEL
LIN {X 0,Y 210.427,Z 433.93,A -85,B 0,C 180,E1 -21152.299,E2 -21152.299} C_VEL
LIN {X 0,Y 212.386,Z 424.213,A -85,B 0,C 180,E1 -21154.507,E2 -21154.507} C_VEL
LIN {X 0,Y 214.471,Z 412.56,A -85,B 0,C 180,E1 -21156.585,E2 -21156.585} C_VEL
LIN {X 0,Y 216.236,Z 401.104,A -85,B 0,C 180,E1 -21158.174,E2 -21158.174} C_VEL
LIN {X 0,Y 217.676,Z 389.366,A -85,B 0,C 180,E1 -21159.407,E2 -21159.407} C_VEL
LIN {X 0,Y 218.969,Z 375.8,A -85,B 0,C 180,E1 -21160.4,E2 -21160.4} C_VEL
LIN {X 0,Y 219.734,Z 362.426,A -85,B 0,C 180,E1 -21161.005,E2 -21161.005} C_VEL
LIN {X 0,Y 222.016,Z 304.069,A -85,B 0,C 180,E1 -21162.837,E2 -21162.837} C_VEL
LIN {X 0,Y 220.643,Z 296.818,A -85,B 0,C 180,E1 -21163.264,E2 -21163.264} C_VEL
LIN {X 0,Y 215.814,Z 282.708,A -85,B 0,C 180,E1 -21164.395,E2 -21164.395} C_VEL
LIN {X 0,Y 209.091,Z 266.541,A -85,B 0,C 180,E1 -21165.936,E2 -21165.936} C_VEL
LIN {X 0,Y 207.116,Z 262.256,A -85,B 0,C 180,E1 -21166.438,E2 -21166.438} C_VEL
LIN {X 0,Y 206.925,Z 261.307,A -85,B 0,C 180,E1 -21166.843,E2 -21166.843} C_VEL
LIN {X 0,Y 206.754,Z 261.226,A -85,B 0,C 180,E1 -21171.956,E2 -21171.956} C_VEL
LIN {X 0,Y 206.701,Z 261.186,A -85,B 0,C 180,E1 -21176.231,E2 -21176.231} C_VEL
LIN {X 0,Y 206.716,Z 261.23,A -85,B 0,C 180,E1 -21180.661,E2 -21180.661} C_VEL
LIN {X 0,Y 206.74,Z 261.214,A -85,B 0,C 180,E1 -21185.346,E2 -21185.346} C_VEL
LIN {X 0,Y 206.726,Z 261.225,A -85,B 0,C 180,E1 -21190.235,E2 -21190.235} C_VEL
LIN {X 0,Y 206.717,Z 261.221,A -85,B 0,C 180,E1 -21194.457,E2 -21194.457} C_VEL
LIN {X 0,Y 206.723,Z 261.226,A -85,B 0,C 180,E1 -21198.411,E2 -21198.411} C_VEL
LIN {X 0,Y 206.701,Z 261.201,A -85,B 0,C 180,E1 -21202.278,E2 -21202.278} C_VEL
LIN {X 0,Y 206.687,Z 261.238,A -85,B 0,C 180,E1 -21207.053,E2 -21207.053} C_VEL
LIN {X 0,Y 206.748,Z 261.184,A -85,B 0,C 180,E1 -21212.105,E2 -21212.105} C_VEL
LIN {X 0,Y 206.78,Z 261.22,A -85,B 0,C 180,E1 -21216.586,E2 -21216.586} C_VEL
LIN {X 0,Y 206.872,Z 261.184,A -85,B 0,C 180,E1 -21222.207,E2 -21222.207} C_VEL
LIN {X 0,Y 206.886,Z 261.167,A -85,B 0,C 180,E1 -21226.253,E2 -21226.253} C_VEL
LIN {X 0,Y 207.125,Z 261.181,A -85,B 0,C 180,E1 -21230.242,E2 -21230.242} C_VEL
LIN {X 0,Y 207.182,Z 261.174,A -85,B 0,C 180,E1 -21232.211,E2 -21232.211} C_VEL
LIN {X 0,Y 207.378,Z 261.098,A -85,B 0,C 180,E1 -21238.067,E2 -21238.067} C_VEL
LIN {X 0,Y 207.509,Z 261.1,A -85,B 0,C 180,E1 -21240.009,E2 -21240.009} C_VEL
LIN {X 0,Y 207.378,Z 261.141,A -85,B 0,C 180,E1 -21241.951,E2 -21241.951} C_VEL
LIN {X 0,Y 207.128,Z 261.157,A -85,B 0,C 180,E1 -21247.809,E2 -21247.809} C_VEL
LIN {X 0,Y 206.926,Z 261.172,A -85,B 0,C 180,E1 -21251.767,E2 -21251.767} C_VEL
LIN {X 0,Y 206.872,Z 261.216,A -85,B 0,C 180,E1 -21255.779,E2 -21255.779} C_VEL
LIN {X 0,Y 206.77,Z 261.197,A -85,B 0,C 180,E1 -21259.879,E2 -21259.879} C_VEL
LIN {X 0,Y 206.756,Z 261.225,A -85,B 0,C 180,E1 -21264.081,E2 -21264.081} C_VEL
LIN {X 0,Y 206.738,Z 261.214,A -85,B 0,C 180,E1 -21268.428,E2 -21268.428} C_VEL
LIN {X 0,Y 206.706,Z 261.238,A -85,B 0,C 180,E1 -21272.965,E2 -21272.965} C_VEL
LIN {X 0,Y 206.686,Z 261.223,A -85,B 0,C 180,E1 -21277.748,E2 -21277.748} C_VEL
LIN {X 0,Y 206.655,Z 261.234,A -85,B 0,C 180,E1 -21281.568,E2 -21281.568} C_VEL
LIN {X 0,Y 206.645,Z 261.191,A -85,B 0,C 180,E1 -21285.588,E2 -21285.588} C_VEL
LIN {X 0,Y 206.648,Z 261.234,A -85,B 0,C 180,E1 -21290.468,E2 -21290.468} C_VEL
LIN {X 0,Y 206.118,Z 261.815,A -85,B 0,C 180,E1 -21291.635,E2 -21291.635} C_VEL
LIN {X 0,Y 204.961,Z 263.342,A -85,B 0,C 180,E1 -21292.72,E2 -21292.72} C_VEL
LIN {X 0,Y 203.428,Z 266.451,A -85,B 0,C 180,E1 -21294.001,E2 -21294.001} C_VEL
LIN {X 0,Y 202.887,Z 269.507,A -85,B 0,C 180,E1 -21294.796,E2 -21294.796} C_VEL
LIN {X 0,Y 203.378,Z 272.735,A -85,B 0,C 180,E1 -21295.313,E2 -21295.313} C_VEL
LIN {X 0,Y 203.489,Z 273.039,A -85,B 0,C 180,E1 -21295.344,E2 -21295.344} C_VEL
LIN {X 0,Y 209.931,Z 289.491,A -85,B 0,C 180,E1 -21296.906,E2 -21296.906} C_VEL
LIN {X 0,Y 213.081,Z 299.091,A -85,B 0,C 180,E1 -21297.696,E2 -21297.696} C_VEL
LIN {X 0,Y 215.185,Z 317.396,A -85,B 0,C 180,E1 -21298.652,E2 -21298.652} C_VEL
LIN {X 0,Y 212.886,Z 375.218,A -85,B 0,C 180,E1 -21300.59,E2 -21300.59} C_VEL
LIN {X 0,Y 211.826,Z 387.376,A -85,B 0,C 180,E1 -21301.312,E2 -21301.312} C_VEL
LIN {X 0,Y 210.409,Z 399.619,A -85,B 0,C 180,E1 -21302.391,E2 -21302.391} C_VEL
LIN {X 0,Y 208.692,Z 411.145,A -85,B 0,C 180,E1 -21303.769,E2 -21303.769} C_VEL
LIN {X 0,Y 206.754,Z 421.644,A -85,B 0,C 180,E1 -21305.393,E2 -21305.393} C_VEL
LIN {X 0,Y 204.981,Z 431.415,A -85,B 0,C 180,E1 -21307.312,E2 -21307.312} C_VEL
LIN {X 0,Y 202.981,Z 441.341,A -85,B 0,C 180,E1 -21309.743,E2 -21309.743} C_VEL
LIN {X 0,Y 201.228,Z 449.451,A -85,B 0,C 180,E1 -21312.207,E2 -21312.207} C_VEL
LIN {X 0,Y 199.572,Z 457.377,A -85,B 0,C 180,E1 -21315.209,E2 -21315.209} C_VEL
LIN {X 0,Y 198.589,Z 462.751,A -85,B 0,C 180,E1 -21317.741,E2 -21317.741} C_VEL
LIN {X 0,Y 197.802,Z 467.969,A -85,B 0,C 180,E1 -21320.8,E2 -21320.8} C_VEL
LIN {X 0,Y 197.36,Z 471.996,A -85,B 0,C 180,E1 -21323.868,E2 -21323.868} C_VEL
LIN {X 0,Y 197.19,Z 474.508,A -85,B 0,C 180,E1 -21326.425,E2 -21326.425} C_VEL
LIN {X 0,Y 197.275,Z 476.927,A -85,B 0,C 180,E1 -21330.001,E2 -21330.001} C_VEL
LIN {X 0,Y 197.199,Z 478.081,A -85,B 0,C 180,E1 -21333.617,E2 -21333.617} C_VEL
LIN {X 0,Y 197.434,Z 478.123,A -85,B 0,C 180,E1 -21336.131,E2 -21336.131} C_VEL
LIN {X 0,Y 198.259,Z 476.995,A -85,B 0,C 180,E1 -21340.21,E2 -21340.21} C_VEL
LIN {X 0,Y 199.961,Z 474.228,A -85,B 0,C 180,E1 -21344.243,E2 -21344.243} C_VEL
LIN {X 0,Y 201.775,Z 471.07,A -85,B 0,C 180,E1 -21347.222,E2 -21347.222} C_VEL
LIN {X 0,Y 204.244,Z 466.877,A -85,B 0,C 180,E1 -21350.127,E2 -21350.127} C_VEL
LIN {X 0,Y 207.709,Z 460.536,A -85,B 0,C 180,E1 -21353.427,E2 -21353.427} C_VEL
LIN {X 0,Y 211.019,Z 453.662,A -85,B 0,C 180,E1 -21356.187,E2 -21356.187} C_VEL
LIN {X 0,Y 215.029,Z 445.063,A -85,B 0,C 180,E1 -21358.822,E2 -21358.822} C_VEL
LIN {X 0,Y 218.762,Z 436.277,A -85,B 0,C 180,E1 -21360.933,E2 -21360.933} C_VEL
LIN {X 0,Y 222.817,Z 425.496,A -85,B 0,C 180,E1 -21362.963,E2 -21362.963} C_VEL
LIN {X 0,Y 226.256,Z 414.665,A -85,B 0,C 180,E1 -21364.534,E2 -21364.534} C_VEL
LIN {X 0,Y 229.415,Z 402.583,A -85,B 0,C 180,E1 -21365.866,E2 -21365.866} C_VEL
LIN {X 0,Y 232.014,Z 389.942,A -85,B 0,C 180,E1 -21366.881,E2 -21366.881} C_VEL
LIN {X 0,Y 233.785,Z 377.2,A -85,B 0,C 180,E1 -21367.582,E2 -21367.582} C_VEL
LIN {X 0,Y 235.139,Z 358.673,A -85,B 0,C 180,E1 -21368.193,E2 -21368.193} C_VEL
LIN {X 0,Y 236.972,Z 326.827,A -85,B 0,C 180,E1 -21369.131,E2 -21369.131} C_VEL
LIN {X 0,Y 231.218,Z 313.806,A -85,B 0,C 180,E1 -21371.225,E2 -21371.225} C_VEL
LIN {X 0,Y 226.372,Z 304.155,A -85,B 0,C 180,E1 -21373.08,E2 -21373.08} C_VEL
LIN {X 0,Y 220.571,Z 294.097,A -85,B 0,C 180,E1 -21375.434,E2 -21375.434} C_VEL
LIN {X 0,Y 216.176,Z 287.014,A -85,B 0,C 180,E1 -21377.382,E2 -21377.382} C_VEL
LIN {X 0,Y 212.61,Z 281.651,A -85,B 0,C 180,E1 -21379.09,E2 -21379.09} C_VEL
LIN {X 0,Y 209.027,Z 276.528,A -85,B 0,C 180,E1 -21380.934,E2 -21380.934} C_VEL
LIN {X 0,Y 204.429,Z 270.215,A -85,B 0,C 180,E1 -21383.542,E2 -21383.542} C_VEL
LIN {X 0,Y 201.405,Z 266.461,A -85,B 0,C 180,E1 -21385.439,E2 -21385.439} C_VEL
LIN {X 0,Y 200.659,Z 264.913,A -85,B 0,C 180,E1 -21386.173,E2 -21386.173} C_VEL
LIN {X 0,Y 199.669,Z 262.14,A -85,B 0,C 180,E1 -21389.449,E2 -21389.449} C_VEL
LIN {X 0,Y 199.647,Z 262.108,A -85,B 0,C 180,E1 -21392.757,E2 -21392.757} C_VEL
LIN {X 0,Y 199.672,Z 262.107,A -85,B 0,C 180,E1 -21397.212,E2 -21397.212} C_VEL
LIN {X 0,Y 199.756,Z 262.099,A -85,B 0,C 180,E1 -21401.795,E2 -21401.795} C_VEL
LIN {X 0,Y 199.823,Z 262.083,A -85,B 0,C 180,E1 -21405.739,E2 -21405.739} C_VEL
LIN {X 0,Y 200.03,Z 262.054,A -85,B 0,C 180,E1 -21409.873,E2 -21409.873} C_VEL
LIN {X 0,Y 200.014,Z 262.054,A -85,B 0,C 180,E1 -21413.94,E2 -21413.94} C_VEL
LIN {X 0,Y 200.294,Z 262.021,A -85,B 0,C 180,E1 -21417.98,E2 -21417.98} C_VEL
LIN {X 0,Y 200.471,Z 262.006,A -85,B 0,C 180,E1 -21419.991,E2 -21419.991} C_VEL
LIN {X 0,Y 200.011,Z 262.059,A -85,B 0,C 180,E1 -21424.021,E2 -21424.021} C_VEL
LIN {X 0,Y 200.072,Z 262.051,A -85,B 0,C 180,E1 -21428.068,E2 -21428.068} C_VEL
LIN {X 0,Y 199.866,Z 262.078,A -85,B 0,C 180,E1 -21432.17,E2 -21432.17} C_VEL
LIN {X 0,Y 199.829,Z 262.346,A -85,B 0,C 180,E1 -21435.284,E2 -21435.284} C_VEL
LIN {X 0,Y 200.307,Z 263.925,A -85,B 0,C 180,E1 -21435.964,E2 -21435.964} C_VEL
LIN {X 0,Y 201.712,Z 266.12,A -85,B 0,C 180,E1 -21436.956,E2 -21436.956} C_VEL
LIN {X 0,Y 204.382,Z 268.396,A -85,B 0,C 180,E1 -21438.536,E2 -21438.536} C_VEL
LIN {X 0,Y 206.422,Z 271.566,A -85,B 0,C 180,E1 -21439.765,E2 -21439.765} C_VEL
LIN {X 0,Y 209.248,Z 274.802,A -85,B 0,C 180,E1 -21441.284,E2 -21441.284} C_VEL
LIN {X 0,Y 213.423,Z 280.575,A -85,B 0,C 180,E1 -21443.404,E2 -21443.404} C_VEL
LIN {X 0,Y 217.329,Z 286.37,A -85,B 0,C 180,E1 -21445.241,E2 -21445.241} C_VEL
LIN {X 0,Y 222.232,Z 294.027,A -85,B 0,C 180,E1 -21447.346,E2 -21447.346} C_VEL
LIN {X 0,Y 227.732,Z 303.542,A -85,B 0,C 180,E1 -21449.528,E2 -21449.528} C_VEL
LIN {X 0,Y 233.918,Z 315.657,A -85,B 0,C 180,E1 -21451.821,E2 -21451.821} C_VEL
LIN {X 0,Y 237.263,Z 323.352,A -85,B 0,C 180,E1 -21453.023,E2 -21453.023} C_VEL
LIN {X 0,Y 234.253,Z 370.284,A -85,B 0,C 180,E1 -21454.412,E2 -21454.412} C_VEL
LIN {X 0,Y 232.544,Z 383.29,A -85,B 0,C 180,E1 -21455.079,E2 -21455.079} C_VEL
LIN {X 0,Y 230.317,Z 395.586,A -85,B 0,C 180,E1 -21456.037,E2 -21456.037} C_VEL
LIN {X 0,Y 227.394,Z 407.303,A -85,B 0,C 180,E1 -21457.264,E2 -21457.264} C_VEL
LIN {X 0,Y 223.938,Z 418.777,A -85,B 0,C 180,E1 -21458.866,E2 -21458.866} C_VEL
LIN {X 0,Y 220.3,Z 429.137,A -85,B 0,C 180,E1 -21460.74,E2 -21460.74} C_VEL
LIN {X 0,Y 216.352,Z 438.848,A -85,B 0,C 180,E1 -21462.999,E2 -21462.999} C_VEL
LIN {X 0,Y 212.623,Z 446.925,A -85,B 0,C 180,E1 -21465.38,E2 -21465.38} C_VEL
LIN {X 0,Y 208.779,Z 454.685,A -85,B 0,C 180,E1 -21468.33,E2 -21468.33} C_VEL
LIN {X 0,Y 205.926,Z 459.835,A -85,B 0,C 180,E1 -21470.847,E2 -21470.847} C_VEL
LIN {X 0,Y 203.081,Z 464.759,A -85,B 0,C 180,E1 -21473.962,E2 -21473.962} C_VEL
LIN {X 0,Y 200.846,Z 468.369,A -85,B 0,C 180,E1 -21477.099,E2 -21477.099} C_VEL
LIN {X 0,Y 199.112,Z 470.928,A -85,B 0,C 180,E1 -21480.385,E2 -21480.385} C_VEL
LIN {X 0,Y 198.268,Z 471.994,A -85,B 0,C 180,E1 -21482.56,E2 -21482.56} C_VEL
LIN {X 0,Y 197.616,Z 472.631,A -85,B 0,C 180,E1 -21484.737,E2 -21484.737} C_VEL
LIN {X 0,Y 197.073,Z 472.735,A -85,B 0,C 180,E1 -21487.972,E2 -21487.972} C_VEL
LIN {X 0,Y 196.794,Z 471.842,A -85,B 0,C 180,E1 -21491.251,E2 -21491.251} C_VEL
LIN {X 0,Y 196.866,Z 469.933,A -85,B 0,C 180,E1 -21494.51,E2 -21494.51} C_VEL
LIN {X 0,Y 197.237,Z 467.071,A -85,B 0,C 180,E1 -21497.655,E2 -21497.655} C_VEL
LIN {X 0,Y 197.806,Z 463.112,A -85,B 0,C 180,E1 -21500.799,E2 -21500.799} C_VEL
LIN {X 0,Y 198.724,Z 457.981,A -85,B 0,C 180,E1 -21503.909,E2 -21503.909} C_VEL
LIN {X 0,Y 199.963,Z 451.526,A -85,B 0,C 180,E1 -21506.977,E2 -21506.977} C_VEL
LIN {X 0,Y 201.56,Z 443.435,A -85,B 0,C 180,E1 -21509.999,E2 -21509.999} C_VEL
LIN {X 0,Y 203.675,Z 433.539,A -85,B 0,C 180,E1 -21512.913,E2 -21512.913} C_VEL
LIN {X 0,Y 205.69,Z 423.877,A -85,B 0,C 180,E1 -21515.145,E2 -21515.145} C_VEL
LIN {X 0,Y 207.835,Z 412.142,A -85,B 0,C 180,E1 -21517.284,E2 -21517.284} C_VEL
LIN {X 0,Y 209.684,Z 400.539,A -85,B 0,C 180,E1 -21518.917,E2 -21518.917} C_VEL
LIN {X 0,Y 211.175,Z 388.53,A -85,B 0,C 180,E1 -21520.183,E2 -21520.183} C_VEL
LIN {X 0,Y 212.443,Z 375.509,A -85,B 0,C 180,E1 -21521.146,E2 -21521.146} C_VEL
LIN {X 0,Y 213.25,Z 361.926,A -85,B 0,C 180,E1 -21521.759,E2 -21521.759} C_VEL
LIN {X 0,Y 215.521,Z 304.596,A -85,B 0,C 180,E1 -21523.615,E2 -21523.615} C_VEL
LIN {X 0,Y 214.301,Z 298.537,A -85,B 0,C 180,E1 -21523.998,E2 -21523.998} C_VEL
LIN {X 0,Y 209.452,Z 284.613,A -85,B 0,C 180,E1 -21525.182,E2 -21525.182} C_VEL
LIN {X 0,Y 202.822,Z 268.587,A -85,B 0,C 180,E1 -21526.773,E2 -21526.773} C_VEL
LIN {X 0,Y 200.043,Z 262.957,A -85,B 0,C 180,E1 -21527.51,E2 -21527.51} C_VEL
LIN {X 0,Y 199.871,Z 262.173,A -85,B 0,C 180,E1 -21527.919,E2 -21527.919} C_VEL
LIN {X 0,Y 199.71,Z 262.09,A -85,B 0,C 180,E1 -21533.828,E2 -21533.828} C_VEL
LIN {X 0,Y 199.684,Z 262.065,A -85,B 0,C 180,E1 -21538.395,E2 -21538.395} C_VEL
LIN {X 0,Y 199.662,Z 262.118,A -85,B 0,C 180,E1 -21542.372,E2 -21542.372} C_VEL
LIN {X 0,Y 199.65,Z 262.105,A -85,B 0,C 180,E1 -21546.756,E2 -21546.756} C_VEL
LIN {X 0,Y 199.693,Z 262.109,A -85,B 0,C 180,E1 -21549.307,E2 -21549.307} C_VEL
LIN {X 0,Y 199.665,Z 262.085,A -85,B 0,C 180,E1 -21552.355,E2 -21552.355} C_VEL
LIN {X 0,Y 199.666,Z 262.109,A -85,B 0,C 180,E1 -21555.269,E2 -21555.269} C_VEL
LIN {X 0,Y 199.671,Z 262.106,A -85,B 0,C 180,E1 -21558.043,E2 -21558.043} C_VEL
LIN {X 0,Y 199.677,Z 262.075,A -85,B 0,C 180,E1 -21560.743,E2 -21560.743} C_VEL
LIN {X 0,Y 199.613,Z 262.118,A -85,B 0,C 180,E1 -21565.726,E2 -21565.726} C_VEL
LIN {X 0,Y 199.683,Z 262.105,A -85,B 0,C 180,E1 -21568.146,E2 -21568.146} C_VEL
LIN {X 0,Y 199.669,Z 262.065,A -85,B 0,C 180,E1 -21572.781,E2 -21572.781} C_VEL
LIN {X 0,Y 199.739,Z 262.103,A -85,B 0,C 180,E1 -21577.24,E2 -21577.24} C_VEL
LIN {X 0,Y 199.825,Z 262.068,A -85,B 0,C 180,E1 -21581.731,E2 -21581.731} C_VEL
LIN {X 0,Y 199.828,Z 262.04,A -85,B 0,C 180,E1 -21585.758,E2 -21585.758} C_VEL
LIN {X 0,Y 200.068,Z 262.06,A -85,B 0,C 180,E1 -21589.894,E2 -21589.894} C_VEL
LIN {X 0,Y 200.125,Z 262.054,A -85,B 0,C 180,E1 -21591.934,E2 -21591.934} C_VEL
LIN {X 0,Y 200.318,Z 261.977,A -85,B 0,C 180,E1 -21597.999,E2 -21597.999} C_VEL
LIN {X 0,Y 200.474,Z 261.976,A -85,B 0,C 180,E1 -21600.009,E2 -21600.009} C_VEL
LIN {X 0,Y 200.02,Z 262.071,A -85,B 0,C 180,E1 -21604.039,E2 -21604.039} C_VEL
LIN {X 0,Y 200.076,Z 262.031,A -85,B 0,C 180,E1 -21608.086,E2 -21608.086} C_VEL
LIN {X 0,Y 199.877,Z 262.054,A -85,B 0,C 180,E1 -21612.188,E2 -21612.188} C_VEL
LIN {X 0,Y 199.81,Z 262.096,A -85,B 0,C 180,E1 -21616.352,E2 -21616.352} C_VEL
LIN {X 0,Y 199.689,Z 262.074,A -85,B 0,C 180,E1 -21620.615,E2 -21620.615} C_VEL
LIN {X 0,Y 199.674,Z 262.114,A -85,B 0,C 180,E1 -21624.993,E2 -21624.993} C_VEL
LIN {X 0,Y 199.639,Z 262.091,A -85,B 0,C 180,E1 -21629.537,E2 -21629.537} C_VEL
LIN {X 0,Y 199.677,Z 262.11,A -85,B 0,C 180,E1 -21632.359,E2 -21632.359} C_VEL
LIN {X 0,Y 199.633,Z 262.101,A -85,B 0,C 180,E1 -21636.77,E2 -21636.77} C_VEL
LIN {X 0,Y 199.619,Z 262.116,A -85,B 0,C 180,E1 -21639.335,E2 -21639.335} C_VEL
LIN {X 0,Y 199.586,Z 262.099,A -85,B 0,C 180,E1 -21642.315,E2 -21642.315} C_VEL
LIN {X 0,Y 199.591,Z 262.068,A -85,B 0,C 180,E1 -21645.233,E2 -21645.233} C_VEL
LIN {X 0,Y 199.584,Z 262.1,A -85,B 0,C 180,E1 -21648.007,E2 -21648.007} C_VEL
LIN {X 0,Y 199.7,Z 262.223,A -85,B 0,C 180,E1 -21652.464,E2 -21652.464} C_VEL
LIN {X 0,Y 200.708,Z 266.357,A -85,B 0,C 180,E1 -21654.554,E2 -21654.554} C_VEL
LIN {X 0,Y 203.176,Z 272.352,A -85,B 0,C 180,E1 -21655.27,E2 -21655.27} C_VEL
LIN {X 0,Y 203.489,Z 273.039,A -85,B 0,C 180,E1 -21655.344,E2 -21655.344} C_VEL
LIN {X 0,Y 205.081,Z 278.505,A -85,B 0,C 180,E1 -21655.796,E2 -21655.796} C_VEL
LIN {X 0,Y 206.267,Z 288.134,A -85,B 0,C 180,E1 -21656.343,E2 -21656.343} C_VEL
LIN {X 0,Y 207.153,Z 303.933,A -85,B 0,C 180,E1 -21657.085,E2 -21657.085} C_VEL
LIN {X 0,Y 208.738,Z 318.396,A -85,B 0,C 180,E1 -21657.862,E2 -21657.862} C_VEL
LIN {X 0,Y 206.444,Z 374.555,A -85,B 0,C 180,E1 -21659.789,E2 -21659.789} C_VEL
LIN {X 0,Y 205.25,Z 387.654,A -85,B 0,C 180,E1 -21660.585,E2 -21660.585} C_VEL
LIN {X 0,Y 203.79,Z 399.803,A -85,B 0,C 180,E1 -21661.694,E2 -21661.694} C_VEL
LIN {X 0,Y 201.993,Z 411.249,A -85,B 0,C 180,E1 -21663.109,E2 -21663.109} C_VEL
LIN {X 0,Y 200.009,Z 421.708,A -85,B 0,C 180,E1 -21664.784,E2 -21664.784} C_VEL
LIN {X 0,Y 198.167,Z 431.452,A -85,B 0,C 180,E1 -21666.763,E2 -21666.763} C_VEL
LIN {X 0,Y 196.194,Z 440.44,A -85,B 0,C 180,E1 -21669.01,E2 -21669.01} C_VEL
LIN {X 0,Y 194.755,Z 447.186,A -85,B 0,C 180,E1 -21671.049,E2 -21671.049} C_VEL
LIN {X 0,Y 192.929,Z 455.515,A -85,B 0,C 180,E1 -21674.145,E2 -21674.145} C_VEL
LIN {X 0,Y 191.633,Z 462.208,A -85,B 0,C 180,E1 -21677.289,E2 -21677.289} C_VEL
LIN {X 0,Y 190.763,Z 467.522,A -85,B 0,C 180,E1 -21680.458,E2 -21680.458} C_VEL
LIN {X 0,Y 190.298,Z 471.633,A -85,B 0,C 180,E1 -21683.64,E2 -21683.64} C_VEL
LIN {X 0,Y 190.091,Z 474.569,A -85,B 0,C 180,E1 -21686.713,E2 -21686.713} C_VEL
LIN {X 0,Y 190.182,Z 476.705,A -85,B 0,C 180,E1 -21690.001,E2 -21690.001} C_VEL
LIN {X 0,Y 190.091,Z 477.838,A -85,B 0,C 180,E1 -21693.286,E2 -21693.286} C_VEL
LIN {X 0,Y 190.379,Z 478.041,A -85,B 0,C 180,E1 -21696.359,E2 -21696.359} C_VEL
LIN {X 0,Y 191.271,Z 476.989,A -85,B 0,C 180,E1 -21700.587,E2 -21700.587} C_VEL
LIN {X 0,Y 192.063,Z 475.871,A -85,B 0,C 180,E1 -21702.683,E2 -21702.683} C_VEL
LIN {X 0,Y 194.25,Z 472.376,A -85,B 0,C 180,E1 -21706.825,E2 -21706.825} C_VEL
LIN {X 0,Y 196.662,Z 468.611,A -85,B 0,C 180,E1 -21709.847,E2 -21709.847} C_VEL
LIN {X 0,Y 199.59,Z 463.755,A -85,B 0,C 180,E1 -21712.789,E2 -21712.789} C_VEL
LIN {X 0,Y 203.196,Z 457.065,A -85,B 0,C 180,E1 -21715.923,E2 -21715.923} C_VEL
LIN {X 0,Y 206.729,Z 450.159,A -85,B 0,C 180,E1 -21718.422,E2 -21718.422} C_VEL
LIN {X 0,Y 210.398,Z 442.485,A -85,B 0,C 180,E1 -21720.625,E2 -21720.625} C_VEL
LIN {X 0,Y 214.809,Z 432.092,A -85,B 0,C 180,E1 -21722.952,E2 -21722.952} C_VEL
LIN {X 0,Y 218.651,Z 421.56,A -85,B 0,C 180,E1 -21724.788,E2 -21724.788} C_VEL
LIN {X 0,Y 222.338,Z 409.731,A -85,B 0,C 180,E1 -21726.348,E2 -21726.348} C_VEL
LIN {X 0,Y 225.462,Z 397.121,A -85,B 0,C 180,E1 -21727.575,E2 -21727.575} C_VEL
LIN {X 0,Y 227.855,Z 384.161,A -85,B 0,C 180,E1 -21728.474,E2 -21728.474} C_VEL
LIN {X 0,Y 229.4,Z 370.411,A -85,B 0,C 180,E1 -21729.086,E2 -21729.086} C_VEL
LIN {X 0,Y 231.915,Z 329.225,A -85,B 0,C 180,E1 -21730.324,E2 -21730.324} C_VEL
LIN {X 0,Y 226.313,Z 316.396,A -85,B 0,C 180,E1 -21732.494,E2 -21732.494} C_VEL
LIN {X 0,Y 221.463,Z 306.809,A -85,B 0,C 180,E1 -21734.47,E2 -21734.47} C_VEL
LIN {X 0,Y 215.32,Z 296.219,A -85,B 0,C 180,E1 -21737.172,E2 -21737.172} C_VEL
LIN {X 0,Y 212.561,Z 291.751,A -85,B 0,C 180,E1 -21738.5,E2 -21738.5} C_VEL
LIN {X 0,Y 209.799,Z 287.479,A -85,B 0,C 180,E1 -21739.898,E2 -21739.898} C_VEL
LIN {X 0,Y 206.32,Z 282.381,A -85,B 0,C 180,E1 -21741.775,E2 -21741.775} C_VEL
LIN {X 0,Y 202.158,Z 276.486,A -85,B 0,C 180,E1 -21744.249,E2 -21744.249} C_VEL
LIN {X 0,Y 199.064,Z 272.479,A -85,B 0,C 180,E1 -21746.283,E2 -21746.283} C_VEL
LIN {X 0,Y 197.964,Z 270.921,A -85,B 0,C 180,E1 -21747.081,E2 -21747.081} C_VEL
LIN {X 0,Y 193.228,Z 265.159,A -85,B 0,C 180,E1 -21750.922,E2 -21750.922} C_VEL
LIN {X 0,Y 192.658,Z 263.376,A -85,B 0,C 180,E1 -21752.862,E2 -21752.862} C_VEL
LIN {X 0,Y 192.564,Z 263.005,A -85,B 0,C 180,E1 -21754.017,E2 -21754.017} C_VEL
LIN {X 0,Y 192.659,Z 262.974,A -85,B 0,C 180,E1 -21756.333,E2 -21756.333} C_VEL
LIN {X 0,Y 192.705,Z 262.973,A -85,B 0,C 180,E1 -21761.484,E2 -21761.484} C_VEL
LIN {X 0,Y 192.748,Z 262.961,A -85,B 0,C 180,E1 -21765.204,E2 -21765.204} C_VEL
LIN {X 0,Y 192.953,Z 262.934,A -85,B 0,C 180,E1 -21769.558,E2 -21769.558} C_VEL
LIN {X 0,Y 192.977,Z 262.931,A -85,B 0,C 180,E1 -21773.718,E2 -21773.718} C_VEL
LIN {X 0,Y 193.239,Z 262.9,A -85,B 0,C 180,E1 -21777.906,E2 -21777.906} C_VEL
LIN {X 0,Y 193.435,Z 262.882,A -85,B 0,C 180,E1 -21779.991,E2 -21779.991} C_VEL
LIN {X 0,Y 192.957,Z 262.939,A -85,B 0,C 180,E1 -21784.168,E2 -21784.168} C_VEL
LIN {X 0,Y 193.023,Z 262.931,A -85,B 0,C 180,E1 -21788.365,E2 -21788.365} C_VEL
LIN {X 0,Y 192.925,Z 263.076,A -85,B 0,C 180,E1 -21790.816,E2 -21790.816} C_VEL
LIN {X 0,Y 193.82,Z 265.787,A -85,B 0,C 180,E1 -21791.884,E2 -21791.884} C_VEL
LIN {X 0,Y 195.791,Z 267.938,A -85,B 0,C 180,E1 -21793.482,E2 -21793.482} C_VEL
LIN {X 0,Y 197.574,Z 268.942,A -85,B 0,C 180,E1 -21794.737,E2 -21794.737} C_VEL
LIN {X 0,Y 199.03,Z 271.777,A -85,B 0,C 180,E1 -21795.872,E2 -21795.872} C_VEL
LIN {X 0,Y 202.003,Z 274.629,A -85,B 0,C 180,E1 -21797.764,E2 -21797.764} C_VEL
LIN {X 0,Y 204.343,Z 278.057,A -85,B 0,C 180,E1 -21799.212,E2 -21799.212} C_VEL
LIN {X 0,Y 206.996,Z 281.294,A -85,B 0,C 180,E1 -21800.696,E2 -21800.696} C_VEL
LIN {X 0,Y 210.629,Z 286.429,A -85,B 0,C 180,E1 -21802.618,E2 -21802.618} C_VEL
LIN {X 0,Y 214.627,Z 292.511,A -85,B 0,C 180,E1 -21804.584,E2 -21804.584} C_VEL
LIN {X 0,Y 221.26,Z 303.451,A -85,B 0,C 180,E1 -21807.524,E2 -21807.524} C_VEL
LIN {X 0,Y 227.236,Z 314.752,A -85,B 0,C 180,E1 -21809.928,E2 -21809.928} C_VEL
LIN {X 0,Y 232.214,Z 325.662,A -85,B 0,C 180,E1 -21811.826,E2 -21811.826} C_VEL
LIN {X 0,Y 229.317,Z 369.818,A -85,B 0,C 180,E1 -21813.15,E2 -21813.15} C_VEL
LIN {X 0,Y 227.572,Z 382.642,A -85,B 0,C 180,E1 -21813.79,E2 -21813.79} C_VEL
LIN {X 0,Y 225.177,Z 395.57,A -85,B 0,C 180,E1 -21814.797,E2 -21814.797} C_VEL
LIN {X 0,Y 221.917,Z 408.137,A -85,B 0,C 180,E1 -21816.14,E2 -21816.14} C_VEL
LIN {X 0,Y 218.113,Z 420.085,A -85,B 0,C 180,E1 -21817.857,E2 -21817.857} C_VEL
LIN {X 0,Y 214.085,Z 430.742,A -85,B 0,C 180,E1 -21819.882,E2 -21819.882} C_VEL
LIN {X 0,Y 210.22,Z 439.72,A -85,B 0,C 180,E1 -21822.072,E2 -21822.072} C_VEL
LIN {X 0,Y 205.808,Z 448.735,A -85,B 0,C 180,E1 -21824.88,E2 -21824.88} C_VEL
LIN {X 0,Y 201.851,Z 456.082,A -85,B 0,C 180,E1 -21827.923,E2 -21827.923} C_VEL
LIN {X 0,Y 198.204,Z 462.185,A -85,B 0,C 180,E1 -21831.251,E2 -21831.251} C_VEL
LIN {X 0,Y 195.194,Z 466.932,A -85,B 0,C 180,E1 -21834.824,E2 -21834.824} C_VEL
LIN {X 0,Y 193.695,Z 469.065,A -85,B 0,C 180,E1 -21837.026,E2 -21837.026} C_VEL
LIN {X 0,Y 192.499,Z 470.738,A -85,B 0,C 180,E1 -21839.26,E2 -21839.26} C_VEL
LIN {X 0,Y 191.414,Z 472.015,A -85,B 0,C 180,E1 -21841.761,E2 -21841.761} C_VEL
LIN {X 0,Y 190.241,Z 472.914,A -85,B 0,C 180,E1 -21846.022,E2 -21846.022} C_VEL
LIN {X 0,Y 189.948,Z 472.748,A -85,B 0,C 180,E1 -21848.284,E2 -21848.284} C_VEL
LIN {X 0,Y 189.714,Z 472.119,A -85,B 0,C 180,E1 -21850.524,E2 -21850.524} C_VEL
LIN {X 0,Y 189.753,Z 470.07,A -85,B 0,C 180,E1 -21854.316,E2 -21854.316} C_VEL
LIN {X 0,Y 190.248,Z 466.499,A -85,B 0,C 180,E1 -21858.277,E2 -21858.277} C_VEL
LIN {X 0,Y 190.895,Z 462.311,A -85,B 0,C 180,E1 -21861.531,E2 -21861.531} C_VEL
LIN {X 0,Y 192.065,Z 455.885,A -85,B 0,C 180,E1 -21865.277,E2 -21865.277} C_VEL
LIN {X 0,Y 193.5,Z 448.893,A -85,B 0,C 180,E1 -21868.438,E2 -21868.438} C_VEL
LIN {X 0,Y 195.035,Z 441.745,A -85,B 0,C 180,E1 -21871.032,E2 -21871.032} C_VEL
LIN {X 0,Y 197.192,Z 431.956,A -85,B 0,C 180,E1 -21873.866,E2 -21873.866} C_VEL
LIN {X 0,Y 199.45,Z 421.172,A -85,B 0,C 180,E1 -21876.321,E2 -21876.321} C_VEL
